    CONST robtarget Target_2200_2:=[[39.025,79.493,0],[0.726314069,0.009187373,0.687236181,-0.009481395],[-2,0,-1,0],[9E+09,9E+09,9E+09,9E+09,9E+09,9E+09]];
    CONST robtarget Target_2210_2:=[[35.542,79.935,0],[0.726314069,0.009187373,0.687236181,-0.009481395],[-2,0,-1,0],[9E+09,9E+09,9E+09,9E+09,9E+09,9E+09]];
    CONST robtarget Target_2220_2:=[[32.97,81.097,0],[0.726314069,0.009187373,0.687236181,-0.009481395],[-2,0,-1,0],[9E+09,9E+09,9E+09,9E+09,9E+09,9E+09]];
    CONST robtarget Target_2230_2:=[[30.756,83.312,0],[0.726314069,0.009187373,0.687236181,-0.009481395],[-2,0,-1,0],[9E+09,9E+09,9E+09,9E+09,9E+09,9E+09]];
    CONST robtarget Target_2240_2:=[[29.841,85.252,0],[0.726314069,0.009187373,0.687236181,-0.009481395],[-2,0,-1,0],[9E+09,9E+09,9E+09,9E+09,9E+09,9E+09]];
    CONST robtarget Target_2250_2:=[[29.28,88.046,0],[0.726314069,0.009187373,0.687236181,-0.009481395],[-2,0,-1,0],[9E+09,9E+09,9E+09,9E+09,9E+09,9E+09]];
    CONST robtarget Target_2260_2:=[[29.205,89.501,0],[0.726314069,0.009187373,0.687236181,-0.009481395],[-2,0,-1,0],[9E+09,9E+09,9E+09,9E+09,9E+09,9E+09]];
    CONST robtarget Target_2270_2:=[[29.324,91.697,0],[0.726314069,0.009187373,0.687236181,-0.009481395],[-2,0,-1,0],[9E+09,9E+09,9E+09,9E+09,9E+09,9E+09]];
    CONST robtarget Target_2280_2:=[[30.172,94.739,0],[0.726314069,0.009187373,0.687236181,-0.009481395],[-2,0,-1,0],[9E+09,9E+09,9E+09,9E+09,9E+09,9E+09]];
    CONST robtarget Target_2290_2:=[[31.657,97.014,0],[0.726314069,0.009187373,0.687236181,-0.009481395],[-2,0,-1,0],[9E+09,9E+09,9E+09,9E+09,9E+09,9E+09]];
    CONST robtarget Target_2300_2:=[[33.883,98.67,0],[0.726314069,0.009187373,0.687236181,-0.009481395],[-2,0,-1,0],[9E+09,9E+09,9E+09,9E+09,9E+09,9E+09]];
    CONST robtarget Target_2310_2:=[[35.769,99.342,0],[0.726314069,0.009187373,0.687236181,-0.009481395],[-2,0,-1,0],[9E+09,9E+09,9E+09,9E+09,9E+09,9E+09]];
    CONST robtarget Target_2320_2:=[[37.808,99.594,0],[0.726314069,0.009187373,0.687236181,-0.009481395],[-2,0,-1,0],[9E+09,9E+09,9E+09,9E+09,9E+09,9E+09]];
    CONST robtarget Target_2330_2:=[[40.664,99.302,0],[0.726314069,0.009187373,0.687236181,-0.009481395],[-2,0,-1,0],[9E+09,9E+09,9E+09,9E+09,9E+09,9E+09]];
    CONST robtarget Target_2340_2:=[[43.731,98.095,0],[0.726314069,0.009187373,0.687236181,-0.009481395],[-2,0,-1,0],[9E+09,9E+09,9E+09,9E+09,9E+09,9E+09]];
    CONST robtarget Target_2350_2:=[[47.413,95.49,0],[0.726314069,0.009187373,0.687236181,-0.009481395],[-2,0,-1,0],[9E+09,9E+09,9E+09,9E+09,9E+09,9E+09]];
    CONST robtarget Target_2360_2:=[[48.093,95.49,0],[0.726314069,0.009187373,0.687236181,-0.009481395],[-2,0,-1,0],[9E+09,9E+09,9E+09,9E+09,9E+09,9E+09]];
    CONST robtarget Target_2370_2:=[[48.093,102.54,0],[0.726314069,0.009187373,0.687236181,-0.009481395],[-2,0,-1,0],[9E+09,9E+09,9E+09,9E+09,9E+09,9E+09]];
    CONST robtarget Target_2380_2:=[[48.093,102.54,10],[0.726314069,0.009187373,0.687236181,-0.009481395],[-2,0,-1,0],[9E+09,9E+09,9E+09,9E+09,9E+09,9E+09]];
    CONST robtarget Target_2390_2:=[[53.685,96.754,10],[0.726314069,0.009187373,0.687236181,-0.009481395],[-2,0,-1,0],[9E+09,9E+09,9E+09,9E+09,9E+09,9E+09]];
    CONST robtarget Target_2400_2:=[[53.685,96.754,0],[0.726314069,0.009187373,0.687236181,-0.009481395],[-2,0,-1,0],[9E+09,9E+09,9E+09,9E+09,9E+09,9E+09]];
    CONST robtarget Target_2410_2:=[[61.781,97.872,0],[0.726314069,0.009187373,0.687236181,-0.009481395],[-2,0,-1,0],[9E+09,9E+09,9E+09,9E+09,9E+09,9E+09]];
    CONST robtarget Target_2420_2:=[[66.233,97.509,0],[0.726314069,0.009187373,0.687236181,-0.009481395],[-2,0,-1,0],[9E+09,9E+09,9E+09,9E+09,9E+09,9E+09]];
    CONST robtarget Target_2430_2:=[[70.243,95.961,0],[0.726314069,0.009187373,0.687236181,-0.009481395],[-2,0,-1,0],[9E+09,9E+09,9E+09,9E+09,9E+09,9E+09]];
    CONST robtarget Target_2440_2:=[[72.614,92.613,0],[0.726314069,0.009187373,0.687236181,-0.009481395],[-2,0,-1,0],[9E+09,9E+09,9E+09,9E+09,9E+09,9E+09]];
    CONST robtarget Target_2450_2:=[[72.964,89.996,0],[0.726314069,0.009187373,0.687236181,-0.009481395],[-2,0,-1,0],[9E+09,9E+09,9E+09,9E+09,9E+09,9E+09]];
    CONST robtarget Target_2460_2:=[[72.964,74.607,0],[0.726314069,0.009187373,0.687236181,-0.009481395],[-2,0,-1,0],[9E+09,9E+09,9E+09,9E+09,9E+09,9E+09]];
    CONST robtarget Target_2470_2:=[[65.962,74.607,0],[0.726314069,0.009187373,0.687236181,-0.009481395],[-2,0,-1,0],[9E+09,9E+09,9E+09,9E+09,9E+09,9E+09]];
    CONST robtarget Target_2480_2:=[[65.962,77.013,0],[0.726314069,0.009187373,0.687236181,-0.009481395],[-2,0,-1,0],[9E+09,9E+09,9E+09,9E+09,9E+09,9E+09]];
    CONST robtarget Target_2490_2:=[[63.118,74.947,0],[0.726314069,0.009187373,0.687236181,-0.009481395],[-2,0,-1,0],[9E+09,9E+09,9E+09,9E+09,9E+09,9E+09]];
    CONST robtarget Target_2500_2:=[[58.766,73.999,0],[0.726314069,0.009187373,0.687236181,-0.009481395],[-2,0,-1,0],[9E+09,9E+09,9E+09,9E+09,9E+09,9E+09]];
    CONST robtarget Target_2510_2:=[[55.832,74.578,0],[0.726314069,0.009187373,0.687236181,-0.009481395],[-2,0,-1,0],[9E+09,9E+09,9E+09,9E+09,9E+09,9E+09]];
    CONST robtarget Target_2520_2:=[[53.483,76.327,0],[0.726314069,0.009187373,0.687236181,-0.009481395],[-2,0,-1,0],[9E+09,9E+09,9E+09,9E+09,9E+09,9E+09]];
    CONST robtarget Target_2530_2:=[[52.081,78.898,0],[0.726314069,0.009187373,0.687236181,-0.009481395],[-2,0,-1,0],[9E+09,9E+09,9E+09,9E+09,9E+09,9E+09]];
    CONST robtarget Target_2540_2:=[[51.789,81.098,0],[0.726314069,0.009187373,0.687236181,-0.009481395],[-2,0,-1,0],[9E+09,9E+09,9E+09,9E+09,9E+09,9E+09]];
    CONST robtarget Target_2550_2:=[[51.983,83.114,0],[0.726314069,0.009187373,0.687236181,-0.009481395],[-2,0,-1,0],[9E+09,9E+09,9E+09,9E+09,9E+09,9E+09]];
    CONST robtarget Target_2560_2:=[[52.864,85.258,0],[0.726314069,0.009187373,0.687236181,-0.009481395],[-2,0,-1,0],[9E+09,9E+09,9E+09,9E+09,9E+09,9E+09]];
    CONST robtarget Target_2570_2:=[[54.039,86.559,0],[0.726314069,0.009187373,0.687236181,-0.009481395],[-2,0,-1,0],[9E+09,9E+09,9E+09,9E+09,9E+09,9E+09]];
    CONST robtarget Target_2580_2:=[[55.703,87.613,0],[0.726314069,0.009187373,0.687236181,-0.009481395],[-2,0,-1,0],[9E+09,9E+09,9E+09,9E+09,9E+09,9E+09]];
    CONST robtarget Target_2590_2:=[[58.542,88.585,0],[0.726314069,0.009187373,0.687236181,-0.009481395],[-2,0,-1,0],[9E+09,9E+09,9E+09,9E+09,9E+09,9E+09]];
    CONST robtarget Target_2600_2:=[[60.612,88.946,0],[0.726314069,0.009187373,0.687236181,-0.009481395],[-2,0,-1,0],[9E+09,9E+09,9E+09,9E+09,9E+09,9E+09]];
    CONST robtarget Target_2610_2:=[[64.587,89.359,0],[0.726314069,0.009187373,0.687236181,-0.009481395],[-2,0,-1,0],[9E+09,9E+09,9E+09,9E+09,9E+09,9E+09]];
    CONST robtarget Target_2620_2:=[[66.011,89.461,0],[0.726314069,0.009187373,0.687236181,-0.009481395],[-2,0,-1,0],[9E+09,9E+09,9E+09,9E+09,9E+09,9E+09]];
    CONST robtarget Target_2630_2:=[[66.011,89.582,0],[0.726314069,0.009187373,0.687236181,-0.009481395],[-2,0,-1,0],[9E+09,9E+09,9E+09,9E+09,9E+09,9E+09]];
    CONST robtarget Target_2640_2:=[[64.625,92.171,0],[0.726314069,0.009187373,0.687236181,-0.009481395],[-2,0,-1,0],[9E+09,9E+09,9E+09,9E+09,9E+09,9E+09]];
    CONST robtarget Target_2650_2:=[[60.468,92.889,0],[0.726314069,0.009187373,0.687236181,-0.009481395],[-2,0,-1,0],[9E+09,9E+09,9E+09,9E+09,9E+09,9E+09]];
    CONST robtarget Target_2660_2:=[[54.293,91.284,0],[0.726314069,0.009187373,0.687236181,-0.009481395],[-2,0,-1,0],[9E+09,9E+09,9E+09,9E+09,9E+09,9E+09]];
    CONST robtarget Target_2670_2:=[[53.685,91.284,0],[0.726314069,0.009187373,0.687236181,-0.009481395],[-2,0,-1,0],[9E+09,9E+09,9E+09,9E+09,9E+09,9E+09]];
    CONST robtarget Target_2680_2:=[[53.685,96.754,0],[0.726314069,0.009187373,0.687236181,-0.009481395],[-2,0,-1,0],[9E+09,9E+09,9E+09,9E+09,9E+09,9E+09]];
    CONST robtarget Target_2690_2:=[[53.685,96.754,10],[0.726314069,0.009187373,0.687236181,-0.009481395],[-2,0,-1,0],[9E+09,9E+09,9E+09,9E+09,9E+09,9E+09]];
    CONST robtarget Target_2700_2:=[[65.962,85.206,10],[0.726314069,0.009187373,0.687236181,-0.009481395],[-2,0,-1,0],[9E+09,9E+09,9E+09,9E+09,9E+09,9E+09]];
    CONST robtarget Target_2710_2:=[[65.962,85.206,0],[0.726314069,0.009187373,0.687236181,-0.009481395],[-2,0,-1,0],[9E+09,9E+09,9E+09,9E+09,9E+09,9E+09]];
    CONST robtarget Target_2720_2:=[[60.881,84.38,0],[0.726314069,0.009187373,0.687236181,-0.009481395],[-2,0,-1,0],[9E+09,9E+09,9E+09,9E+09,9E+09,9E+09]];
    CONST robtarget Target_2730_2:=[[59.422,83.407,0],[0.726314069,0.009187373,0.687236181,-0.009481395],[-2,0,-1,0],[9E+09,9E+09,9E+09,9E+09,9E+09,9E+09]];
    CONST robtarget Target_2740_2:=[[58.912,81.681,0],[0.726314069,0.009187373,0.687236181,-0.009481395],[-2,0,-1,0],[9E+09,9E+09,9E+09,9E+09,9E+09,9E+09]];
    CONST robtarget Target_2750_2:=[[59.032,80.639,0],[0.726314069,0.009187373,0.687236181,-0.009481395],[-2,0,-1,0],[9E+09,9E+09,9E+09,9E+09,9E+09,9E+09]];
    CONST robtarget Target_2760_2:=[[60.054,79.339,0],[0.726314069,0.009187373,0.687236181,-0.009481395],[-2,0,-1,0],[9E+09,9E+09,9E+09,9E+09,9E+09,9E+09]];
    CONST robtarget Target_2770_2:=[[61.465,78.954,0],[0.726314069,0.009187373,0.687236181,-0.009481395],[-2,0,-1,0],[9E+09,9E+09,9E+09,9E+09,9E+09,9E+09]];
    CONST robtarget Target_2780_2:=[[62.315,78.91,0],[0.726314069,0.009187373,0.687236181,-0.009481395],[-2,0,-1,0],[9E+09,9E+09,9E+09,9E+09,9E+09,9E+09]];
    CONST robtarget Target_2790_2:=[[64.212,79.335,0],[0.726314069,0.009187373,0.687236181,-0.009481395],[-2,0,-1,0],[9E+09,9E+09,9E+09,9E+09,9E+09,9E+09]];
    CONST robtarget Target_2800_2:=[[65.962,80.514,0],[0.726314069,0.009187373,0.687236181,-0.009481395],[-2,0,-1,0],[9E+09,9E+09,9E+09,9E+09,9E+09,9E+09]];
    CONST robtarget Target_2810_2:=[[65.962,85.206,0],[0.726314069,0.009187373,0.687236181,-0.009481395],[-2,0,-1,0],[9E+09,9E+09,9E+09,9E+09,9E+09,9E+09]];
    CONST robtarget Target_2820_2:=[[65.962,85.206,10],[0.726314069,0.009187373,0.687236181,-0.009481395],[-2,0,-1,0],[9E+09,9E+09,9E+09,9E+09,9E+09,9E+09]];
    CONST robtarget Target_2830_2:=[[78.191,105.944,10],[0.726314069,0.009187373,0.687236181,-0.009481395],[-2,0,-1,0],[9E+09,9E+09,9E+09,9E+09,9E+09,9E+09]];
    CONST robtarget Target_2840_2:=[[78.191,105.944,0],[0.726314069,0.009187373,0.687236181,-0.009481395],[-2,0,-1,0],[9E+09,9E+09,9E+09,9E+09,9E+09,9E+09]];
    CONST robtarget Target_2850_2:=[[78.191,74.607,0],[0.726314069,0.009187373,0.687236181,-0.009481395],[-2,0,-1,0],[9E+09,9E+09,9E+09,9E+09,9E+09,9E+09]];
    CONST robtarget Target_2860_2:=[[84.949,74.607,0],[0.726314069,0.009187373,0.687236181,-0.009481395],[-1,0,-1,0],[9E+09,9E+09,9E+09,9E+09,9E+09,9E+09]];
    CONST robtarget Target_2870_2:=[[85.241,75.725,0],[0.726314069,0.009187373,0.687236181,-0.009481395],[-1,0,-1,0],[9E+09,9E+09,9E+09,9E+09,9E+09,9E+09]];
    CONST robtarget Target_2880_2:=[[90.832,74.169,0],[0.726314069,0.009187373,0.687236181,-0.009481395],[-1,0,-1,0],[9E+09,9E+09,9E+09,9E+09,9E+09,9E+09]];
    CONST robtarget Target_2890_2:=[[94.512,74.978,0],[0.726314069,0.009187373,0.687236181,-0.009481395],[-1,0,-1,0],[9E+09,9E+09,9E+09,9E+09,9E+09,9E+09]];
    CONST robtarget Target_2900_2:=[[97.536,77.39,0],[0.726314069,0.009187373,0.687236181,-0.009481395],[-1,-1,0,0],[9E+09,9E+09,9E+09,9E+09,9E+09,9E+09]];
    CONST robtarget Target_2910_2:=[[99.251,80.187,0],[0.726314069,0.009187373,0.687236181,-0.009481395],[-1,-1,0,0],[9E+09,9E+09,9E+09,9E+09,9E+09,9E+09]];
    CONST robtarget Target_2920_2:=[[100.173,83.531,0],[0.726314069,0.009187373,0.687236181,-0.009481395],[-1,-1,0,0],[9E+09,9E+09,9E+09,9E+09,9E+09,9E+09]];
    CONST robtarget Target_2930_2:=[[100.362,86.227,0],[0.726314069,0.009187373,0.687236181,-0.009481395],[-1,-1,0,0],[9E+09,9E+09,9E+09,9E+09,9E+09,9E+09]];
    CONST robtarget Target_2940_2:=[[100.162,89.348,0],[0.726314069,0.009187373,0.687236181,-0.009481395],[-1,-1,0,0],[9E+09,9E+09,9E+09,9E+09,9E+09,9E+09]];
    CONST robtarget Target_2950_2:=[[99.451,92.348,0],[0.726314069,0.009187373,0.687236181,-0.009481395],[-1,-1,0,0],[9E+09,9E+09,9E+09,9E+09,9E+09,9E+09]];
    CONST robtarget Target_2960_2:=[[98.126,94.909,0],[0.726314069,0.009187373,0.687236181,-0.009481395],[-1,-1,0,0],[9E+09,9E+09,9E+09,9E+09,9E+09,9E+09]];
    CONST robtarget Target_2970_2:=[[96.145,96.789,0],[0.726314069,0.009187373,0.687236181,-0.009481395],[-1,0,-1,0],[9E+09,9E+09,9E+09,9E+09,9E+09,9E+09]];
    CONST robtarget Target_2980_2:=[[93.246,97.782,0],[0.726314069,0.009187373,0.687236181,-0.009481395],[-1,0,-1,0],[9E+09,9E+09,9E+09,9E+09,9E+09,9E+09]];
    CONST robtarget Target_2990_2:=[[91.056,97.792,0],[0.726314069,0.009187373,0.687236181,-0.009481395],[-1,0,-1,0],[9E+09,9E+09,9E+09,9E+09,9E+09,9E+09]];
    CONST robtarget Target_3000_2:=[[88.708,97.17,0],[0.726314069,0.009187373,0.687236181,-0.009481395],[-1,0,-1,0],[9E+09,9E+09,9E+09,9E+09,9E+09,9E+09]];
    CONST robtarget Target_3010_2:=[[86.849,96.094,0],[0.726314069,0.009187373,0.687236181,-0.009481395],[-1,0,-1,0],[9E+09,9E+09,9E+09,9E+09,9E+09,9E+09]];
    CONST robtarget Target_3020_2:=[[85.241,94.858,0],[0.726314069,0.009187373,0.687236181,-0.009481395],[-1,0,-1,0],[9E+09,9E+09,9E+09,9E+09,9E+09,9E+09]];
    CONST robtarget Target_3030_2:=[[85.241,105.944,0],[0.726314069,0.009187373,0.687236181,-0.009481395],[-1,0,-1,0],[9E+09,9E+09,9E+09,9E+09,9E+09,9E+09]];
    CONST robtarget Target_3040_2:=[[78.191,105.944,0],[0.726314069,0.009187373,0.687236181,-0.009481395],[-2,0,-1,0],[9E+09,9E+09,9E+09,9E+09,9E+09,9E+09]];
    CONST robtarget Target_3050_2:=[[78.191,105.944,10],[0.726314069,0.009187373,0.687236181,-0.009481395],[-2,0,-1,0],[9E+09,9E+09,9E+09,9E+09,9E+09,9E+09]];
    CONST robtarget Target_3060_2:=[[85.241,91.138,10],[0.726314069,0.009187373,0.687236181,-0.009481395],[-1,0,-1,0],[9E+09,9E+09,9E+09,9E+09,9E+09,9E+09]];
    CONST robtarget Target_3070_2:=[[85.241,91.138,0],[0.726314069,0.009187373,0.687236181,-0.009481395],[-1,0,-1,0],[9E+09,9E+09,9E+09,9E+09,9E+09,9E+09]];
    CONST robtarget Target_3080_2:=[[85.241,79.809,0],[0.726314069,0.009187373,0.687236181,-0.009481395],[-1,0,-1,0],[9E+09,9E+09,9E+09,9E+09,9E+09,9E+09]];
    CONST robtarget Target_3090_2:=[[88.085,79.323,0],[0.726314069,0.009187373,0.687236181,-0.009481395],[-1,0,-1,0],[9E+09,9E+09,9E+09,9E+09,9E+09,9E+09]];
    CONST robtarget Target_3100_2:=[[90.106,79.66,0],[0.726314069,0.009187373,0.687236181,-0.009481395],[-1,0,-1,0],[9E+09,9E+09,9E+09,9E+09,9E+09,9E+09]];
    CONST robtarget Target_3110_2:=[[91.905,81.033,0],[0.726314069,0.009187373,0.687236181,-0.009481395],[-1,0,-1,0],[9E+09,9E+09,9E+09,9E+09,9E+09,9E+09]];
    CONST robtarget Target_3120_2:=[[92.891,83.394,0],[0.726314069,0.009187373,0.687236181,-0.009481395],[-1,0,-1,0],[9E+09,9E+09,9E+09,9E+09,9E+09,9E+09]];
    CONST robtarget Target_3130_2:=[[93.142,86.082,0],[0.726314069,0.009187373,0.687236181,-0.009481395],[-1,0,-1,0],[9E+09,9E+09,9E+09,9E+09,9E+09,9E+09]];
    CONST robtarget Target_3140_2:=[[92.957,88.611,0],[0.726314069,0.009187373,0.687236181,-0.009481395],[-1,0,-1,0],[9E+09,9E+09,9E+09,9E+09,9E+09,9E+09]];
    CONST robtarget Target_3150_2:=[[92.311,90.605,0],[0.726314069,0.009187373,0.687236181,-0.009481395],[-1,0,-1,0],[9E+09,9E+09,9E+09,9E+09,9E+09,9E+09]];
    CONST robtarget Target_3160_2:=[[90.724,92.035,0],[0.726314069,0.009187373,0.687236181,-0.009481395],[-1,0,-1,0],[9E+09,9E+09,9E+09,9E+09,9E+09,9E+09]];
    CONST robtarget Target_3170_2:=[[88.961,92.354,0],[0.726314069,0.009187373,0.687236181,-0.009481395],[-1,0,-1,0],[9E+09,9E+09,9E+09,9E+09,9E+09,9E+09]];
    CONST robtarget Target_3180_2:=[[87.176,92.081,0],[0.726314069,0.009187373,0.687236181,-0.009481395],[-1,0,-1,0],[9E+09,9E+09,9E+09,9E+09,9E+09,9E+09]];
    CONST robtarget Target_3190_2:=[[85.241,91.138,0],[0.726314069,0.009187373,0.687236181,-0.009481395],[-1,0,-1,0],[9E+09,9E+09,9E+09,9E+09,9E+09,9E+09]];
    CONST robtarget Target_3200_2:=[[85.241,91.138,10],[0.726314069,0.009187373,0.687236181,-0.009481395],[-1,0,-1,0],[9E+09,9E+09,9E+09,9E+09,9E+09,9E+09]];
    CONST robtarget Target_3210_2:=[[114.293,92.889,10],[0.726314069,0.009187373,0.687236181,-0.009481395],[-1,-1,0,0],[9E+09,9E+09,9E+09,9E+09,9E+09,9E+09]];
    CONST robtarget Target_3220_2:=[[114.293,92.889,0],[0.726314069,0.009187373,0.687236181,-0.009481395],[-1,-1,0,0],[9E+09,9E+09,9E+09,9E+09,9E+09,9E+09]];
    CONST robtarget Target_3230_2:=[[111.516,91.894,0],[0.726314069,0.009187373,0.687236181,-0.009481395],[-1,-1,0,0],[9E+09,9E+09,9E+09,9E+09,9E+09,9E+09]];
    CONST robtarget Target_3240_2:=[[110.079,88.878,0],[0.726314069,0.009187373,0.687236181,-0.009481395],[-1,-1,0,0],[9E+09,9E+09,9E+09,9E+09,9E+09,9E+09]];
    CONST robtarget Target_3250_2:=[[109.82,85.731,0],[0.726314069,0.009187373,0.687236181,-0.009481395],[-1,-1,0,0],[9E+09,9E+09,9E+09,9E+09,9E+09,9E+09]];
    CONST robtarget Target_3260_2:=[[110.134,82.622,0],[0.726314069,0.009187373,0.687236181,-0.009481395],[-1,-1,0,0],[9E+09,9E+09,9E+09,9E+09,9E+09,9E+09]];
    CONST robtarget Target_3270_2:=[[112.748,79.215,0],[0.726314069,0.009187373,0.687236181,-0.009481395],[-1,-1,0,0],[9E+09,9E+09,9E+09,9E+09,9E+09,9E+09]];
    CONST robtarget Target_3280_2:=[[115.472,79.116,0],[0.726314069,0.009187373,0.687236181,-0.009481395],[-1,-1,0,0],[9E+09,9E+09,9E+09,9E+09,9E+09,9E+09]];
    CONST robtarget Target_3290_2:=[[117.853,81.029,0],[0.726314069,0.009187373,0.687236181,-0.009481395],[-1,-1,0,0],[9E+09,9E+09,9E+09,9E+09,9E+09,9E+09]];
    CONST robtarget Target_3300_2:=[[118.692,84.329,0],[0.726314069,0.009187373,0.687236181,-0.009481395],[-1,-1,0,0],[9E+09,9E+09,9E+09,9E+09,9E+09,9E+09]];
    CONST robtarget Target_3310_2:=[[118.705,87.144,0],[0.726314069,0.009187373,0.687236181,-0.009481395],[-1,-1,0,0],[9E+09,9E+09,9E+09,9E+09,9E+09,9E+09]];
    CONST robtarget Target_3320_2:=[[117.699,91.082,0],[0.726314069,0.009187373,0.687236181,-0.009481395],[-1,-1,0,0],[9E+09,9E+09,9E+09,9E+09,9E+09,9E+09]];
    CONST robtarget Target_3330_2:=[[116.9,92.042,0],[0.726314069,0.009187373,0.687236181,-0.009481395],[-1,-1,0,0],[9E+09,9E+09,9E+09,9E+09,9E+09,9E+09]];
    CONST robtarget Target_3340_2:=[[114.293,92.889,0],[0.726314069,0.009187373,0.687236181,-0.009481395],[-1,-1,0,0],[9E+09,9E+09,9E+09,9E+09,9E+09,9E+09]];
    CONST robtarget Target_3350_2:=[[114.293,92.889,10],[0.726314069,0.009187373,0.687236181,-0.009481395],[-1,-1,0,0],[9E+09,9E+09,9E+09,9E+09,9E+09,9E+09]];
    CONST robtarget Target_3360_2:=[[114.293,97.945,10],[0.726314069,0.009187373,0.687236181,-0.009481395],[-1,-1,0,0],[9E+09,9E+09,9E+09,9E+09,9E+09,9E+09]];
    CONST robtarget Target_3370_2:=[[114.293,97.945,0],[0.726314069,0.009187373,0.687236181,-0.009481395],[-1,-1,0,0],[9E+09,9E+09,9E+09,9E+09,9E+09,9E+09]];
    CONST robtarget Target_3380_2:=[[119.425,97.063,0],[0.726314069,0.009187373,0.687236181,-0.009481395],[-1,-1,0,0],[9E+09,9E+09,9E+09,9E+09,9E+09,9E+09]];
    CONST robtarget Target_3390_2:=[[122.854,94.783,0],[0.726314069,0.009187373,0.687236181,-0.009481395],[-1,-1,0,0],[9E+09,9E+09,9E+09,9E+09,9E+09,9E+09]];
    CONST robtarget Target_3400_2:=[[124.981,91.496,0],[0.726314069,0.009187373,0.687236181,-0.009481395],[-1,-1,0,0],[9E+09,9E+09,9E+09,9E+09,9E+09,9E+09]];
    CONST robtarget Target_3410_2:=[[125.918,87.222,0],[0.726314069,0.009187373,0.687236181,-0.009481395],[-1,-1,0,0],[9E+09,9E+09,9E+09,9E+09,9E+09,9E+09]];
    CONST robtarget Target_3420_2:=[[125.74,83.065,0],[0.726314069,0.009187373,0.687236181,-0.009481395],[-1,-1,0,0],[9E+09,9E+09,9E+09,9E+09,9E+09,9E+09]];
    CONST robtarget Target_3430_2:=[[124.292,78.941,0],[0.726314069,0.009187373,0.687236181,-0.009481395],[-1,-1,0,0],[9E+09,9E+09,9E+09,9E+09,9E+09,9E+09]];
    CONST robtarget Target_3440_2:=[[122.614,76.811,0],[0.726314069,0.009187373,0.687236181,-0.009481395],[-1,-1,0,0],[9E+09,9E+09,9E+09,9E+09,9E+09,9E+09]];
    CONST robtarget Target_3450_2:=[[118.869,74.576,0],[0.726314069,0.009187373,0.687236181,-0.009481395],[-1,-1,0,0],[9E+09,9E+09,9E+09,9E+09,9E+09,9E+09]];
    CONST robtarget Target_3460_2:=[[115.671,73.954,0],[0.726314069,0.009187373,0.687236181,-0.009481395],[-1,-1,0,0],[9E+09,9E+09,9E+09,9E+09,9E+09,9E+09]];
    CONST robtarget Target_3470_2:=[[111.694,74.099,0],[0.726314069,0.009187373,0.687236181,-0.009481395],[-1,-1,0,0],[9E+09,9E+09,9E+09,9E+09,9E+09,9E+09]];
    CONST robtarget Target_3480_2:=[[107.574,75.575,0],[0.726314069,0.009187373,0.687236181,-0.009481395],[-1,-1,0,0],[9E+09,9E+09,9E+09,9E+09,9E+09,9E+09]];
    CONST robtarget Target_3490_2:=[[104.577,78.476,0],[0.726314069,0.009187373,0.687236181,-0.009481395],[-1,-1,0,0],[9E+09,9E+09,9E+09,9E+09,9E+09,9E+09]];
    CONST robtarget Target_3500_2:=[[103.102,81.78,0],[0.726314069,0.009187373,0.687236181,-0.009481395],[-1,-1,0,0],[9E+09,9E+09,9E+09,9E+09,9E+09,9E+09]];
    CONST robtarget Target_3510_2:=[[102.673,84.234,0],[0.726314069,0.009187373,0.687236181,-0.009481395],[-1,-1,0,0],[9E+09,9E+09,9E+09,9E+09,9E+09,9E+09]];
    CONST robtarget Target_3520_2:=[[102.712,87.979,0],[0.726314069,0.009187373,0.687236181,-0.009481395],[-1,-1,0,0],[9E+09,9E+09,9E+09,9E+09,9E+09,9E+09]];
    CONST robtarget Target_3530_2:=[[103.395,91.017,0],[0.726314069,0.009187373,0.687236181,-0.009481395],[-1,-1,0,0],[9E+09,9E+09,9E+09,9E+09,9E+09,9E+09]];
    CONST robtarget Target_3540_2:=[[104.511,93.286,0],[0.726314069,0.009187373,0.687236181,-0.009481395],[-1,-1,0,0],[9E+09,9E+09,9E+09,9E+09,9E+09,9E+09]];
    CONST robtarget Target_3550_2:=[[106.651,95.634,0],[0.726314069,0.009187373,0.687236181,-0.009481395],[-1,-1,0,0],[9E+09,9E+09,9E+09,9E+09,9E+09,9E+09]];
    CONST robtarget Target_3560_2:=[[109.412,97.163,0],[0.726314069,0.009187373,0.687236181,-0.009481395],[-1,-1,0,0],[9E+09,9E+09,9E+09,9E+09,9E+09,9E+09]];
    CONST robtarget Target_3570_2:=[[114.293,97.945,0],[0.726314069,0.009187373,0.687236181,-0.009481395],[-1,-1,0,0],[9E+09,9E+09,9E+09,9E+09,9E+09,9E+09]];
    CONST robtarget Target_3580_2:=[[114.293,97.945,10],[0.726314069,0.009187373,0.687236181,-0.009481395],[-1,-1,0,0],[9E+09,9E+09,9E+09,9E+09,9E+09,9E+09]];
    CONST robtarget Target_3590_2:=[[57.132,66.1,10],[0.726314069,0.009187373,0.687236181,-0.009481395],[-2,0,-1,0],[9E+09,9E+09,9E+09,9E+09,9E+09,9E+09]];
    CONST robtarget Target_3600_2:=[[57.132,66.1,0],[0.726314069,0.009187373,0.687236181,-0.009481395],[-2,0,-1,0],[9E+09,9E+09,9E+09,9E+09,9E+09,9E+09]];
    CONST robtarget Target_3610_2:=[[40.852,48.713,0],[0.726314069,0.009187373,0.687236181,-0.009481395],[-2,0,-1,0],[9E+09,9E+09,9E+09,9E+09,9E+09,9E+09]];
    CONST robtarget Target_3620_2:=[[40.852,45.296,0],[0.726314069,0.009187373,0.687236181,-0.009481395],[-2,0,-1,0],[9E+09,9E+09,9E+09,9E+09,9E+09,9E+09]];
    CONST robtarget Target_3630_2:=[[75,4.113,0],[0.726314069,0.009187373,0.687236181,-0.009481395],[-2,0,-1,0],[9E+09,9E+09,9E+09,9E+09,9E+09,9E+09]];
    CONST robtarget Target_3640_2:=[[109.148,45.296,0],[0.726314069,0.009187373,0.687236181,-0.009481395],[-1,-1,0,0],[9E+09,9E+09,9E+09,9E+09,9E+09,9E+09]];
    CONST robtarget Target_3650_2:=[[109.148,48.713,0],[0.726314069,0.009187373,0.687236181,-0.009481395],[-1,-1,0,0],[9E+09,9E+09,9E+09,9E+09,9E+09,9E+09]];
    CONST robtarget Target_3660_2:=[[92.868,66.1,0],[0.726314069,0.009187373,0.687236181,-0.009481395],[-1,0,-1,0],[9E+09,9E+09,9E+09,9E+09,9E+09,9E+09]];
    CONST robtarget Target_3670_2:=[[57.132,66.1,0],[0.726314069,0.009187373,0.687236181,-0.009481395],[-2,0,-1,0],[9E+09,9E+09,9E+09,9E+09,9E+09,9E+09]];
    CONST robtarget Target_3680_2:=[[57.132,66.1,10],[0.726314069,0.009187373,0.687236181,-0.009481395],[-2,0,-1,0],[9E+09,9E+09,9E+09,9E+09,9E+09,9E+09]];
    CONST robtarget Target_3690_2:=[[59.3,61.1,10],[0.726314069,0.009187373,0.687236181,-0.009481395],[-2,0,-1,0],[9E+09,9E+09,9E+09,9E+09,9E+09,9E+09]];
    CONST robtarget Target_3700_2:=[[59.3,61.1,0],[0.726314069,0.009187373,0.687236181,-0.009481395],[-2,0,-1,0],[9E+09,9E+09,9E+09,9E+09,9E+09,9E+09]];
    CONST robtarget Target_3710_2:=[[48.446,49.508,0],[0.726314069,0.009187373,0.687236181,-0.009481395],[-2,0,-1,0],[9E+09,9E+09,9E+09,9E+09,9E+09,9E+09]];
    CONST robtarget Target_3720_2:=[[59.481,49.508,0],[0.726314069,0.009187373,0.687236181,-0.009481395],[-2,0,-1,0],[9E+09,9E+09,9E+09,9E+09,9E+09,9E+09]];
    CONST robtarget Target_3730_2:=[[69.526,61.1,0],[0.726314069,0.009187373,0.687236181,-0.009481395],[-2,0,-1,0],[9E+09,9E+09,9E+09,9E+09,9E+09,9E+09]];
    CONST robtarget Target_3740_2:=[[59.3,61.1,0],[0.726314069,0.009187373,0.687236181,-0.009481395],[-2,0,-1,0],[9E+09,9E+09,9E+09,9E+09,9E+09,9E+09]];
    CONST robtarget Target_3750_2:=[[59.3,61.1,10],[0.726314069,0.009187373,0.687236181,-0.009481395],[-2,0,-1,0],[9E+09,9E+09,9E+09,9E+09,9E+09,9E+09]];
    CONST robtarget Target_3760_2:=[[80.474,61.1,10],[0.726314069,0.009187373,0.687236181,-0.009481395],[-2,0,-1,0],[9E+09,9E+09,9E+09,9E+09,9E+09,9E+09]];
    CONST robtarget Target_3770_2:=[[80.474,61.1,0],[0.726314069,0.009187373,0.687236181,-0.009481395],[-2,0,-1,0],[9E+09,9E+09,9E+09,9E+09,9E+09,9E+09]];
    CONST robtarget Target_3780_2:=[[90.7,61.1,0],[0.726314069,0.009187373,0.687236181,-0.009481395],[-1,0,-1,0],[9E+09,9E+09,9E+09,9E+09,9E+09,9E+09]];
    CONST robtarget Target_3790_2:=[[101.554,49.508,0],[0.726314069,0.009187373,0.687236181,-0.009481395],[-1,-1,0,0],[9E+09,9E+09,9E+09,9E+09,9E+09,9E+09]];
    CONST robtarget Target_3800_2:=[[90.519,49.508,0],[0.726314069,0.009187373,0.687236181,-0.009481395],[-1,0,-1,0],[9E+09,9E+09,9E+09,9E+09,9E+09,9E+09]];
    CONST robtarget Target_3810_2:=[[80.474,61.1,0],[0.726314069,0.009187373,0.687236181,-0.009481395],[-2,0,-1,0],[9E+09,9E+09,9E+09,9E+09,9E+09,9E+09]];
    CONST robtarget Target_3820_2:=[[80.474,61.1,10],[0.726314069,0.009187373,0.687236181,-0.009481395],[-2,0,-1,0],[9E+09,9E+09,9E+09,9E+09,9E+09,9E+09]];
    CONST robtarget Target_3830_2:=[[75,59.782,10],[0.726314069,0.009187373,0.687236181,-0.009481395],[-2,0,-1,0],[9E+09,9E+09,9E+09,9E+09,9E+09,9E+09]];
    CONST robtarget Target_3840_2:=[[75,59.782,0],[0.726314069,0.009187373,0.687236181,-0.009481395],[-2,0,-1,0],[9E+09,9E+09,9E+09,9E+09,9E+09,9E+09]];
    CONST robtarget Target_3850_2:=[[83.903,49.508,0],[0.726314069,0.009187373,0.687236181,-0.009481395],[-1,0,-1,0],[9E+09,9E+09,9E+09,9E+09,9E+09,9E+09]];
    CONST robtarget Target_3860_2:=[[66.097,49.508,0],[0.726314069,0.009187373,0.687236181,-0.009481395],[-2,0,-1,0],[9E+09,9E+09,9E+09,9E+09,9E+09,9E+09]];
    CONST robtarget Target_3870_2:=[[75,59.782,0],[0.726314069,0.009187373,0.687236181,-0.009481395],[-2,0,-1,0],[9E+09,9E+09,9E+09,9E+09,9E+09,9E+09]];
    CONST robtarget Target_3880_2:=[[75,59.782,10],[0.726314069,0.009187373,0.687236181,-0.009481395],[-2,0,-1,0],[9E+09,9E+09,9E+09,9E+09,9E+09,9E+09]];
    CONST robtarget Target_3890_2:=[[64.21,44.508,10],[0.726314069,0.009187373,0.687236181,-0.009481395],[-2,0,-1,0],[9E+09,9E+09,9E+09,9E+09,9E+09,9E+09]];
    CONST robtarget Target_3900_2:=[[64.21,44.508,0],[0.726314069,0.009187373,0.687236181,-0.009481395],[-2,0,-1,0],[9E+09,9E+09,9E+09,9E+09,9E+09,9E+09]];
    CONST robtarget Target_3910_2:=[[85.79,44.508,0],[0.726314069,0.009187373,0.687236181,-0.009481395],[-1,0,-1,0],[9E+09,9E+09,9E+09,9E+09,9E+09,9E+09]];
    CONST robtarget Target_3920_2:=[[75,15.254,0],[0.726314069,0.009187373,0.687236181,-0.009481395],[-2,0,-1,0],[9E+09,9E+09,9E+09,9E+09,9E+09,9E+09]];
    CONST robtarget Target_3930_2:=[[64.21,44.508,0],[0.726314069,0.009187373,0.687236181,-0.009481395],[-2,0,-1,0],[9E+09,9E+09,9E+09,9E+09,9E+09,9E+09]];
    CONST robtarget Target_3940_2:=[[64.21,44.508,10],[0.726314069,0.009187373,0.687236181,-0.009481395],[-2,0,-1,0],[9E+09,9E+09,9E+09,9E+09,9E+09,9E+09]];
    CONST robtarget Target_3950_2:=[[58.88,44.508,10],[0.726314069,0.009187373,0.687236181,-0.009481395],[-2,0,-1,0],[9E+09,9E+09,9E+09,9E+09,9E+09,9E+09]];
    CONST robtarget Target_3960_2:=[[58.88,44.508,0],[0.726314069,0.009187373,0.687236181,-0.009481395],[-2,0,-1,0],[9E+09,9E+09,9E+09,9E+09,9E+09,9E+09]];
    CONST robtarget Target_3970_2:=[[48.001,44.508,0],[0.726314069,0.009187373,0.687236181,-0.009481395],[-2,0,-1,0],[9E+09,9E+09,9E+09,9E+09,9E+09,9E+09]];
    CONST robtarget Target_3980_2:=[[67.598,20.874,0],[0.726314069,0.009187373,0.687236181,-0.009481395],[-2,0,-1,0],[9E+09,9E+09,9E+09,9E+09,9E+09,9E+09]];
    CONST robtarget Target_3990_2:=[[58.88,44.508,0],[0.726314069,0.009187373,0.687236181,-0.009481395],[-2,0,-1,0],[9E+09,9E+09,9E+09,9E+09,9E+09,9E+09]];
    CONST robtarget Target_4000_2:=[[58.88,44.508,10],[0.726314069,0.009187373,0.687236181,-0.009481395],[-2,0,-1,0],[9E+09,9E+09,9E+09,9E+09,9E+09,9E+09]];
    CONST robtarget Target_4010_2:=[[91.12,44.508,10],[0.726314069,0.009187373,0.687236181,-0.009481395],[-1,0,-1,0],[9E+09,9E+09,9E+09,9E+09,9E+09,9E+09]];
    CONST robtarget Target_4020_2:=[[91.12,44.508,0],[0.726314069,0.009187373,0.687236181,-0.009481395],[-1,0,-1,0],[9E+09,9E+09,9E+09,9E+09,9E+09,9E+09]];
    CONST robtarget Target_4030_2:=[[101.999,44.508,0],[0.726314069,0.009187373,0.687236181,-0.009481395],[-1,-1,0,0],[9E+09,9E+09,9E+09,9E+09,9E+09,9E+09]];
    CONST robtarget Target_4040_2:=[[82.402,20.874,0],[0.726314069,0.009187373,0.687236181,-0.009481395],[-1,0,-1,0],[9E+09,9E+09,9E+09,9E+09,9E+09,9E+09]];
    CONST robtarget Target_4050_2:=[[91.12,44.508,0],[0.726314069,0.009187373,0.687236181,-0.009481395],[-1,0,-1,0],[9E+09,9E+09,9E+09,9E+09,9E+09,9E+09]];
    CONST robtarget Target_Home_Espejo:=[[-676.754166789,677.141454372,-133.14230978],[0.358218118,-0.604139007,0.620387065,0.349021104],[-1,0,-1,0],[9E+09,9E+09,9E+09,9E+09,9E+09,9E+09]];
!Ejercicio hecho en clase
    !TASK PERS wobjdata wcaja:=[FALSE,TRUE,"",[[-78.3768,-694.538,672.47],[0.999913,-0.00011372,0.00016022,0.0132033]],[[-74.9038,-552.314,679.445],[0.0262226,-0.999656,6.92619E-06,1.8063E-05]]];
    !***********************************************************
    !
    ! M?dulo:  Module1
    !
    ! Descripción:
    !   <Introduzca la descripción aquí>
    !
    ! Autor: GabrielBojaca y Mafe Morillo
    !
    ! Versión: 1.0
    !
    !***********************************************************


    !***********************************************************
    !
    ! Procedimiento Main
    !
    !   Este es el punto de entrada de su programa
    !
    !***********************************************************
    PROC main()
        !MoveAbsJ Home_ABS, v1000, z1, tool0;
        !Path_10;
        MoveAbsJ Home_ABS, v300, z1, tool0;

        TPErase;
        TPWrite "INICIO PROGRAMA";
        TPWrite "APAGADO BANDA TRANASPORTADORA";
        Reset DO_02;
        Reset DO_01;
        RESET BWD_Conveyor;
        RESET FWD_Conveyor;

        WHILE TRUE DO
            IF DI_03 = 1 THEN
                RESET BWD_Conveyor;
                Reset FWD_Conveyor;
                Set BWD_Conveyor;
                WaitTime 2;
                Reset FWD_Conveyor;
                Reset BWD_Conveyor;
            ENDIF

            IF DI_01 = 1 AND DI_02 = 0 THEN
                TPWrite "ENCIENDE BANDA TRANASPORTADORA";
                Set FWD_Conveyor;
                WaitTime 2.03;  !2.05 el mejor hasta ahora
                TPWrite "APAGADO BANDA TRANASPORTADORA";
                Reset FWD_Conveyor;
                TPWrite "INICIANDO DECORADO";
                Set DO_01;
                Path_10;
                TPWrite "DECORADO FINALIZADO";
                Reset DO_01;
                MoveAbsJ Home_ABS,v1000,z1,tool0;
                TPWrite "ENCENDIDO BANDA TRANASPORTADORA";
                Set FWD_Conveyor;
                WaitTime 8;
                TPWrite "APAGADO BANDA TRANASPORTADORA";
                Reset FWD_Conveyor;

            ELSEIF DI_01 = 0 AND DI_02=1 THEN
                Set DO_02;
                TPWrite "RUTINA CAMBIO DE HERRAMIENTA";
                MoveAbsJ Mantenimiento_Point,v1000,z1,tool0;
                TPWrite "PELIGRO";
                TPWrite "OPERARIO CERCA A HERRAMIENTA";
                TPWrite "PRESIONE LOS DOS BOTONES PARA CONTINUAR EL PROGRAMA";
                WaitDI DI_01,1;
                WaitDI DI_02,1;
                Reset DO_02;
                TPWrite "REANUDANDO PROGRAMA";
                WaitTime 3;
                MoveAbsJ Home_ABS,v1000,z1,tool0;
            ELSEIF DI_01 = 0 AND DI_02=0 THEN
                TPWrite "ESPERANDO INSTRUCCIÓNES";
            ELSEIF DI_01 = 1 AND DI_02=1 THEN
                TPWrite "ERROR";
                TPWrite "NO DEBE PRESIONAR AMBAS ENTRADAS AL TIEMPO";
            ENDIF

        ENDWHILE



    ENDPROC

    PROC Test_Caja()
        RESET BWD_Conveyor;
        Reset FWD_Conveyor;
        Set BWD_Conveyor;
        WaitTime 2;
        Reset FWD_Conveyor;
        Reset BWD_Conveyor;
    ENDPROC

    PROC Aristas_Caja()
        MoveL Target_10,v1000,z1,Marcador_TCP\WObj:=Caja;
        MoveL Target_20,v1000,z1,Marcador_TCP\WObj:=Caja;
        MoveL Target_30,v1000,z1,Marcador_TCP\WObj:=Caja;
        MoveL Target_40,v1000,z1,Marcador_TCP\WObj:=Caja;
    ENDPROC
    PROC MAFE()

    ENDPROC
    PROC Path_10()
        MoveL Home_cafe,v1000,z1,Marcador_TCP\WObj:=Caja;
        MoveL Target_60,v1000,z1,Marcador_TCP\WObj:=Caja;
        MoveL Target_70,v1000,z1,Marcador_TCP\WObj:=Caja;
        MoveL Target_80,v1000,z1,Marcador_TCP\WObj:=Caja;
        MoveL Target_90,v1000,z1,Marcador_TCP\WObj:=Caja;
        MoveL Target_100,v1000,z1,Marcador_TCP\WObj:=Caja;
        MoveL Target_110,v1000,z1,Marcador_TCP\WObj:=Caja;
        MoveL Target_120,v1000,z1,Marcador_TCP\WObj:=Caja;
        MoveL Target_130,v1000,z1,Marcador_TCP\WObj:=Caja;
        MoveL Target_140,v1000,z1,Marcador_TCP\WObj:=Caja;
        MoveL Target_150,v1000,z1,Marcador_TCP\WObj:=Caja;
        MoveL Target_160,v1000,z1,Marcador_TCP\WObj:=Caja;
        MoveL Target_170,v1000,z1,Marcador_TCP\WObj:=Caja;
        MoveL Target_180,v1000,z1,Marcador_TCP\WObj:=Caja;
        MoveL Target_190,v1000,z1,Marcador_TCP\WObj:=Caja;
        MoveL Target_200,v1000,z1,Marcador_TCP\WObj:=Caja;
        MoveL Target_210,v1000,z1,Marcador_TCP\WObj:=Caja;
        MoveL Target_220,v1000,z1,Marcador_TCP\WObj:=Caja;
        MoveL Target_230,v1000,z1,Marcador_TCP\WObj:=Caja;
        MoveL Target_240,v1000,z1,Marcador_TCP\WObj:=Caja;
        MoveL Target_250,v1000,z1,Marcador_TCP\WObj:=Caja;
        MoveL Target_260,v1000,z1,Marcador_TCP\WObj:=Caja;
        MoveL Target_270,v1000,z1,Marcador_TCP\WObj:=Caja;
        MoveL Target_280,v1000,z1,Marcador_TCP\WObj:=Caja;
        MoveL Target_290,v1000,z1,Marcador_TCP\WObj:=Caja;
        MoveL Target_300,v1000,z1,Marcador_TCP\WObj:=Caja;
        MoveL Target_310,v1000,z1,Marcador_TCP\WObj:=Caja;
        MoveL Target_320,v1000,z1,Marcador_TCP\WObj:=Caja;
        MoveL Target_330,v1000,z1,Marcador_TCP\WObj:=Caja;
        MoveL Target_340,v1000,z1,Marcador_TCP\WObj:=Caja;
        MoveL Target_350,v1000,z1,Marcador_TCP\WObj:=Caja;
        MoveL Target_360,v1000,z1,Marcador_TCP\WObj:=Caja;
        MoveL Target_370,v1000,z1,Marcador_TCP\WObj:=Caja;
        MoveL Target_380,v1000,z1,Marcador_TCP\WObj:=Caja;
        MoveL Target_390,v1000,z1,Marcador_TCP\WObj:=Caja;
        MoveL Target_400,v1000,z1,Marcador_TCP\WObj:=Caja;
        MoveL Target_410,v1000,z1,Marcador_TCP\WObj:=Caja;
        MoveL Target_420,v1000,z1,Marcador_TCP\WObj:=Caja;
        MoveL Target_430,v1000,z1,Marcador_TCP\WObj:=Caja;
        MoveL Target_440,v1000,z1,Marcador_TCP\WObj:=Caja;
        MoveL Target_450,v1000,z1,Marcador_TCP\WObj:=Caja;
        MoveL Target_460,v1000,z1,Marcador_TCP\WObj:=Caja;
        MoveL Target_470,v1000,z1,Marcador_TCP\WObj:=Caja;
        MoveL Target_480,v1000,z1,Marcador_TCP\WObj:=Caja;
        MoveL Target_490,v1000,z1,Marcador_TCP\WObj:=Caja;
        MoveL Target_500,v1000,z1,Marcador_TCP\WObj:=Caja;
        MoveL Target_510,v1000,z1,Marcador_TCP\WObj:=Caja;
        MoveL Target_520,v1000,z1,Marcador_TCP\WObj:=Caja;
        MoveL Target_530,v1000,z1,Marcador_TCP\WObj:=Caja;
        MoveL Target_540,v1000,z1,Marcador_TCP\WObj:=Caja;
        MoveL Target_550,v1000,z1,Marcador_TCP\WObj:=Caja;
        MoveL Target_560,v1000,z1,Marcador_TCP\WObj:=Caja;
        MoveL Target_570,v1000,z1,Marcador_TCP\WObj:=Caja;
        MoveL Target_580,v1000,z1,Marcador_TCP\WObj:=Caja;
        MoveL Target_590,v1000,z1,Marcador_TCP\WObj:=Caja;
        MoveL Target_600,v1000,z1,Marcador_TCP\WObj:=Caja;
        MoveL Target_610,v1000,z1,Marcador_TCP\WObj:=Caja;
        MoveL Target_620,v1000,z1,Marcador_TCP\WObj:=Caja;
        MoveL Target_630,v1000,z1,Marcador_TCP\WObj:=Caja;
        MoveL Target_640,v1000,z1,Marcador_TCP\WObj:=Caja;
        MoveL Target_650,v1000,z1,Marcador_TCP\WObj:=Caja;
        MoveL Target_660,v1000,z1,Marcador_TCP\WObj:=Caja;
        MoveL Target_670,v1000,z1,Marcador_TCP\WObj:=Caja;
        MoveL Target_680,v1000,z1,Marcador_TCP\WObj:=Caja;
        MoveL Target_690,v1000,z1,Marcador_TCP\WObj:=Caja;
        MoveL Target_700,v1000,z1,Marcador_TCP\WObj:=Caja;
        MoveL Target_710,v1000,z1,Marcador_TCP\WObj:=Caja;
        MoveL Target_720,v1000,z1,Marcador_TCP\WObj:=Caja;
        MoveL Target_730,v1000,z1,Marcador_TCP\WObj:=Caja;
        MoveL Target_740,v1000,z1,Marcador_TCP\WObj:=Caja;
        MoveL Target_750,v1000,z1,Marcador_TCP\WObj:=Caja;
        MoveL Target_760,v1000,z1,Marcador_TCP\WObj:=Caja;
        MoveL Target_770,v1000,z1,Marcador_TCP\WObj:=Caja;
        MoveL Target_780,v1000,z1,Marcador_TCP\WObj:=Caja;
        MoveL Target_790,v1000,z1,Marcador_TCP\WObj:=Caja;
        MoveL Target_800,v1000,z1,Marcador_TCP\WObj:=Caja;
        MoveL Target_810,v1000,z1,Marcador_TCP\WObj:=Caja;
        MoveL Target_820,v1000,z1,Marcador_TCP\WObj:=Caja;
        MoveL Target_830,v1000,z1,Marcador_TCP\WObj:=Caja;
        MoveL Target_840,v1000,z1,Marcador_TCP\WObj:=Caja;
        MoveL Target_850,v1000,z1,Marcador_TCP\WObj:=Caja;
        MoveL Target_860,v1000,z1,Marcador_TCP\WObj:=Caja;
        MoveL Target_870,v1000,z1,Marcador_TCP\WObj:=Caja;
        MoveL Target_880,v1000,z1,Marcador_TCP\WObj:=Caja;
        MoveL Target_890,v1000,z1,Marcador_TCP\WObj:=Caja;
        MoveL Target_900,v1000,z1,Marcador_TCP\WObj:=Caja;
        MoveL Target_910,v1000,z1,Marcador_TCP\WObj:=Caja;
        MoveL Target_920,v1000,z1,Marcador_TCP\WObj:=Caja;
        MoveL Target_930,v1000,z1,Marcador_TCP\WObj:=Caja;
        MoveL Target_940,v1000,z1,Marcador_TCP\WObj:=Caja;
        MoveL Target_950,v1000,z1,Marcador_TCP\WObj:=Caja;
        MoveL Target_960,v1000,z1,Marcador_TCP\WObj:=Caja;
        MoveL Target_970,v1000,z1,Marcador_TCP\WObj:=Caja;
        MoveL Target_980,v1000,z1,Marcador_TCP\WObj:=Caja;
        MoveL Target_990,v1000,z1,Marcador_TCP\WObj:=Caja;
        MoveL Target_1000,v1000,z1,Marcador_TCP\WObj:=Caja;
        MoveL Target_1010,v1000,z1,Marcador_TCP\WObj:=Caja;
        MoveL Target_1020,v1000,z1,Marcador_TCP\WObj:=Caja;
        MoveL Target_1030,v1000,z1,Marcador_TCP\WObj:=Caja;
        MoveL Target_1040,v1000,z1,Marcador_TCP\WObj:=Caja;
        MoveL Target_1050,v1000,z1,Marcador_TCP\WObj:=Caja;
        MoveL Target_1060,v1000,z1,Marcador_TCP\WObj:=Caja;
        MoveL Target_1070,v1000,z1,Marcador_TCP\WObj:=Caja;
        MoveL Target_1080,v1000,z1,Marcador_TCP\WObj:=Caja;
        MoveL Target_1090,v1000,z1,Marcador_TCP\WObj:=Caja;
        MoveL Target_1100,v1000,z1,Marcador_TCP\WObj:=Caja;
        MoveL Target_1110,v1000,z1,Marcador_TCP\WObj:=Caja;
        MoveL Target_1120,v1000,z1,Marcador_TCP\WObj:=Caja;
        MoveL Target_1130,v1000,z1,Marcador_TCP\WObj:=Caja;
        MoveL Target_1140,v1000,z1,Marcador_TCP\WObj:=Caja;
        MoveL Target_1150,v1000,z1,Marcador_TCP\WObj:=Caja;
        MoveL Target_1160,v1000,z1,Marcador_TCP\WObj:=Caja;
        MoveL Target_1170,v1000,z1,Marcador_TCP\WObj:=Caja;
        MoveL Target_1180,v1000,z1,Marcador_TCP\WObj:=Caja;
        MoveL Target_1190,v1000,z1,Marcador_TCP\WObj:=Caja;
        MoveL Target_1200,v1000,z1,Marcador_TCP\WObj:=Caja;
        MoveL Target_1210,v1000,z1,Marcador_TCP\WObj:=Caja;
        MoveL Target_1220,v1000,z1,Marcador_TCP\WObj:=Caja;
        MoveL Target_1230,v1000,z1,Marcador_TCP\WObj:=Caja;
        MoveL Target_1240,v1000,z1,Marcador_TCP\WObj:=Caja;
        MoveL Target_1250,v1000,z1,Marcador_TCP\WObj:=Caja;
        MoveL Target_1260,v1000,z1,Marcador_TCP\WObj:=Caja;
        MoveL Target_1270,v1000,z1,Marcador_TCP\WObj:=Caja;
        MoveL Target_1280,v1000,z1,Marcador_TCP\WObj:=Caja;
        MoveL Target_1290,v1000,z1,Marcador_TCP\WObj:=Caja;
        MoveL Target_1300,v1000,z1,Marcador_TCP\WObj:=Caja;
        MoveL Target_1310,v1000,z1,Marcador_TCP\WObj:=Caja;
        MoveL Target_1320,v1000,z1,Marcador_TCP\WObj:=Caja;
        MoveL Target_1330,v1000,z1,Marcador_TCP\WObj:=Caja;
        MoveL Target_1340,v1000,z1,Marcador_TCP\WObj:=Caja;
        MoveL Target_1350,v1000,z1,Marcador_TCP\WObj:=Caja;
        MoveL Target_1360,v1000,z1,Marcador_TCP\WObj:=Caja;
        MoveL Target_1370,v1000,z1,Marcador_TCP\WObj:=Caja;
        MoveL Target_1380,v1000,z1,Marcador_TCP\WObj:=Caja;
        MoveL Target_1390,v1000,z1,Marcador_TCP\WObj:=Caja;
        MoveL Target_1400,v1000,z1,Marcador_TCP\WObj:=Caja;
        MoveL Target_1410,v1000,z1,Marcador_TCP\WObj:=Caja;
        MoveL Target_1420,v1000,z1,Marcador_TCP\WObj:=Caja;
        MoveL Target_1430,v1000,z1,Marcador_TCP\WObj:=Caja;
        MoveL Target_1440,v1000,z1,Marcador_TCP\WObj:=Caja;
        MoveL Target_1450,v1000,z1,Marcador_TCP\WObj:=Caja;
        MoveL Target_1460,v1000,z1,Marcador_TCP\WObj:=Caja;
        MoveL Target_1470,v1000,z1,Marcador_TCP\WObj:=Caja;
        MoveL Target_1480,v1000,z1,Marcador_TCP\WObj:=Caja;
        MoveL Target_1490,v1000,z1,Marcador_TCP\WObj:=Caja;
        MoveL Target_1500,v1000,z1,Marcador_TCP\WObj:=Caja;
        MoveL Target_1510,v1000,z1,Marcador_TCP\WObj:=Caja;
        MoveL Target_1520,v1000,z1,Marcador_TCP\WObj:=Caja;
        MoveL Target_1530,v1000,z1,Marcador_TCP\WObj:=Caja;
        MoveL Target_1540,v1000,z1,Marcador_TCP\WObj:=Caja;
        MoveL Target_1550,v1000,z1,Marcador_TCP\WObj:=Caja;
        MoveL Target_1560,v1000,z1,Marcador_TCP\WObj:=Caja;
        MoveL Target_1570,v1000,z1,Marcador_TCP\WObj:=Caja;
        MoveL Target_1580,v1000,z1,Marcador_TCP\WObj:=Caja;
        MoveL Target_1590,v1000,z1,Marcador_TCP\WObj:=Caja;
        MoveL Target_1600,v1000,z1,Marcador_TCP\WObj:=Caja;
        MoveL Target_1610,v1000,z1,Marcador_TCP\WObj:=Caja;
        MoveL Target_1620,v1000,z1,Marcador_TCP\WObj:=Caja;
        MoveL Target_1630,v1000,z1,Marcador_TCP\WObj:=Caja;
        MoveL Target_1640,v1000,z1,Marcador_TCP\WObj:=Caja;
        MoveL Target_1650,v1000,z1,Marcador_TCP\WObj:=Caja;
        MoveL Target_1660,v1000,z1,Marcador_TCP\WObj:=Caja;
        MoveL Target_1670,v1000,z1,Marcador_TCP\WObj:=Caja;
        MoveL Target_1680,v1000,z1,Marcador_TCP\WObj:=Caja;
        MoveL Target_1690,v1000,z1,Marcador_TCP\WObj:=Caja;
        MoveL Target_1700,v1000,z1,Marcador_TCP\WObj:=Caja;
        MoveL Target_1710,v1000,z1,Marcador_TCP\WObj:=Caja;
        MoveL Target_1720,v1000,z1,Marcador_TCP\WObj:=Caja;
        MoveL Target_1730,v1000,z1,Marcador_TCP\WObj:=Caja;
        MoveL Target_1740,v1000,z1,Marcador_TCP\WObj:=Caja;
        MoveL Target_1750,v1000,z1,Marcador_TCP\WObj:=Caja;
        MoveL Target_1760,v1000,z1,Marcador_TCP\WObj:=Caja;
        MoveL Target_1770,v1000,z1,Marcador_TCP\WObj:=Caja;
        MoveL Target_1780,v1000,z1,Marcador_TCP\WObj:=Caja;
        MoveL Target_1790,v1000,z1,Marcador_TCP\WObj:=Caja;
        MoveL Target_1800,v1000,z1,Marcador_TCP\WObj:=Caja;
        MoveL Target_1810,v1000,z1,Marcador_TCP\WObj:=Caja;
        MoveL Target_1820,v1000,z1,Marcador_TCP\WObj:=Caja;
        MoveL Target_1830,v1000,z1,Marcador_TCP\WObj:=Caja;
        MoveL Target_1840,v1000,z1,Marcador_TCP\WObj:=Caja;
        MoveL Target_1850,v1000,z1,Marcador_TCP\WObj:=Caja;
        MoveL Target_1860,v1000,z1,Marcador_TCP\WObj:=Caja;
        MoveL Target_1870,v1000,z1,Marcador_TCP\WObj:=Caja;
        MoveL Target_1880,v1000,z1,Marcador_TCP\WObj:=Caja;
        MoveL Target_1890,v1000,z1,Marcador_TCP\WObj:=Caja;
        MoveL Target_1900,v1000,z1,Marcador_TCP\WObj:=Caja;
        MoveL Target_1910,v1000,z1,Marcador_TCP\WObj:=Caja;
        MoveL Target_1920,v1000,z1,Marcador_TCP\WObj:=Caja;
        MoveL Target_1930,v1000,z1,Marcador_TCP\WObj:=Caja;
        MoveL Target_1940,v1000,z1,Marcador_TCP\WObj:=Caja;
        MoveL Target_1950,v1000,z1,Marcador_TCP\WObj:=Caja;
        MoveL Target_1960,v1000,z1,Marcador_TCP\WObj:=Caja;
        MoveL Target_1970,v1000,z1,Marcador_TCP\WObj:=Caja;
        MoveL Target_1980,v1000,z1,Marcador_TCP\WObj:=Caja;
        MoveL Target_1990,v1000,z1,Marcador_TCP\WObj:=Caja;
        MoveL Target_2000,v1000,z1,Marcador_TCP\WObj:=Caja;
        MoveL Target_2010,v1000,z1,Marcador_TCP\WObj:=Caja;
        MoveL Target_2020,v1000,z1,Marcador_TCP\WObj:=Caja;
        MoveL Target_2030,v1000,z1,Marcador_TCP\WObj:=Caja;
        MoveL Target_2040,v1000,z1,Marcador_TCP\WObj:=Caja;
        MoveL Target_2050,v1000,z1,Marcador_TCP\WObj:=Caja;
        MoveL Target_2060,v1000,z1,Marcador_TCP\WObj:=Caja;
        MoveL Target_2070,v1000,z1,Marcador_TCP\WObj:=Caja;
        MoveL Target_2080,v1000,z1,Marcador_TCP\WObj:=Caja;
        MoveL Target_2090,v1000,z1,Marcador_TCP\WObj:=Caja;
        MoveL Target_2100,v1000,z1,Marcador_TCP\WObj:=Caja;
        MoveL Target_2110,v1000,z1,Marcador_TCP\WObj:=Caja;
        MoveL Target_2120,v1000,z1,Marcador_TCP\WObj:=Caja;
        MoveL Target_2130,v1000,z1,Marcador_TCP\WObj:=Caja;
        MoveL Target_2140,v1000,z1,Marcador_TCP\WObj:=Caja;
        MoveL Target_2150,v1000,z1,Marcador_TCP\WObj:=Caja;
        MoveL Target_2160,v1000,z1,Marcador_TCP\WObj:=Caja;
        MoveL Target_2170,v1000,z1,Marcador_TCP\WObj:=Caja;
        MoveL Target_2180,v1000,z1,Marcador_TCP\WObj:=Caja;
        MoveL Target_2190,v1000,z1,Marcador_TCP\WObj:=Caja;
        MoveL Target_2200,v1000,z1,Marcador_TCP\WObj:=Caja;
        MoveL Target_2210,v1000,z1,Marcador_TCP\WObj:=Caja;
        MoveL Target_2220,v1000,z1,Marcador_TCP\WObj:=Caja;
        MoveL Target_2230,v1000,z1,Marcador_TCP\WObj:=Caja;
        MoveL Target_2240,v1000,z1,Marcador_TCP\WObj:=Caja;
        MoveL Target_2250,v1000,z1,Marcador_TCP\WObj:=Caja;
        MoveL Target_2260,v1000,z1,Marcador_TCP\WObj:=Caja;
        MoveL Target_2270,v1000,z1,Marcador_TCP\WObj:=Caja;
        MoveL Target_2280,v1000,z1,Marcador_TCP\WObj:=Caja;
        MoveL Target_2290,v1000,z1,Marcador_TCP\WObj:=Caja;
        MoveL Target_2300,v1000,z1,Marcador_TCP\WObj:=Caja;
        MoveL Target_2310,v1000,z1,Marcador_TCP\WObj:=Caja;
        MoveL Target_2320,v1000,z1,Marcador_TCP\WObj:=Caja;
        MoveL Target_2330,v1000,z1,Marcador_TCP\WObj:=Caja;
        MoveL Target_2340,v1000,z1,Marcador_TCP\WObj:=Caja;
        MoveL Target_2350,v1000,z1,Marcador_TCP\WObj:=Caja;
        MoveL Target_2360,v1000,z1,Marcador_TCP\WObj:=Caja;
        MoveL Target_2370,v1000,z1,Marcador_TCP\WObj:=Caja;
        MoveL Target_2380,v1000,z1,Marcador_TCP\WObj:=Caja;
        MoveL Target_2390,v1000,z1,Marcador_TCP\WObj:=Caja;
        MoveL Target_2400,v1000,z1,Marcador_TCP\WObj:=Caja;
        MoveL Target_2410,v1000,z1,Marcador_TCP\WObj:=Caja;
        MoveL Target_2420,v1000,z1,Marcador_TCP\WObj:=Caja;
        MoveL Target_2430,v1000,z1,Marcador_TCP\WObj:=Caja;
        MoveL Target_2440,v1000,z1,Marcador_TCP\WObj:=Caja;
        MoveL Target_2450,v1000,z1,Marcador_TCP\WObj:=Caja;
        MoveL Target_2460,v1000,z1,Marcador_TCP\WObj:=Caja;
        MoveL Target_2470,v1000,z1,Marcador_TCP\WObj:=Caja;
        MoveL Target_2480,v1000,z1,Marcador_TCP\WObj:=Caja;
        MoveL Target_2490,v1000,z1,Marcador_TCP\WObj:=Caja;
        MoveL Target_2500,v1000,z1,Marcador_TCP\WObj:=Caja;
        MoveL Target_2510,v1000,z1,Marcador_TCP\WObj:=Caja;
        MoveL Target_2520,v1000,z1,Marcador_TCP\WObj:=Caja;
        MoveL Target_2530,v1000,z1,Marcador_TCP\WObj:=Caja;
        MoveL Target_2540,v1000,z1,Marcador_TCP\WObj:=Caja;
        MoveL Target_2550,v1000,z1,Marcador_TCP\WObj:=Caja;
        MoveL Target_2560,v1000,z1,Marcador_TCP\WObj:=Caja;
        MoveL Target_2570,v1000,z1,Marcador_TCP\WObj:=Caja;
        MoveL Target_2580,v1000,z1,Marcador_TCP\WObj:=Caja;
        MoveL Target_2590,v1000,z1,Marcador_TCP\WObj:=Caja;
        MoveL Target_2600,v1000,z1,Marcador_TCP\WObj:=Caja;
        MoveL Target_2610,v1000,z1,Marcador_TCP\WObj:=Caja;
        MoveL Target_2620,v1000,z1,Marcador_TCP\WObj:=Caja;
        MoveL Target_2630,v1000,z1,Marcador_TCP\WObj:=Caja;
        MoveL Target_2640,v1000,z1,Marcador_TCP\WObj:=Caja;
        MoveL Target_2650,v1000,z1,Marcador_TCP\WObj:=Caja;
        MoveL Target_2660,v1000,z1,Marcador_TCP\WObj:=Caja;
        MoveL Target_2670,v1000,z1,Marcador_TCP\WObj:=Caja;
        MoveL Target_2680,v1000,z1,Marcador_TCP\WObj:=Caja;
        MoveL Target_2690,v1000,z1,Marcador_TCP\WObj:=Caja;
        MoveL Target_2700,v1000,z1,Marcador_TCP\WObj:=Caja;
        MoveL Target_2710,v1000,z1,Marcador_TCP\WObj:=Caja;
        MoveL Target_2720,v1000,z1,Marcador_TCP\WObj:=Caja;
        MoveL Target_2730,v1000,z1,Marcador_TCP\WObj:=Caja;
        MoveL Target_2740,v1000,z1,Marcador_TCP\WObj:=Caja;
        MoveL Target_2750,v1000,z1,Marcador_TCP\WObj:=Caja;
        MoveL Target_2760,v1000,z1,Marcador_TCP\WObj:=Caja;
        MoveL Target_2770,v1000,z1,Marcador_TCP\WObj:=Caja;
        MoveL Target_2780,v1000,z1,Marcador_TCP\WObj:=Caja;
        MoveL Target_2790,v1000,z1,Marcador_TCP\WObj:=Caja;
        MoveL Target_2800,v1000,z1,Marcador_TCP\WObj:=Caja;
        MoveL Target_2810,v1000,z1,Marcador_TCP\WObj:=Caja;
        MoveL Target_2820,v1000,z1,Marcador_TCP\WObj:=Caja;
        MoveL Target_2830,v1000,z1,Marcador_TCP\WObj:=Caja;
        MoveL Target_2840,v1000,z1,Marcador_TCP\WObj:=Caja;
        MoveL Target_2850,v1000,z1,Marcador_TCP\WObj:=Caja;
        MoveL Target_2860,v1000,z1,Marcador_TCP\WObj:=Caja;
        MoveL Target_2870,v1000,z1,Marcador_TCP\WObj:=Caja;
        MoveL Target_2880,v1000,z1,Marcador_TCP\WObj:=Caja;
        MoveL Target_2890,v1000,z1,Marcador_TCP\WObj:=Caja;
        MoveL Target_2900,v1000,z1,Marcador_TCP\WObj:=Caja;
        MoveL Target_2910,v1000,z1,Marcador_TCP\WObj:=Caja;
        MoveL Target_2920,v1000,z1,Marcador_TCP\WObj:=Caja;
        MoveL Target_2930,v1000,z1,Marcador_TCP\WObj:=Caja;
        MoveL Target_2940,v1000,z1,Marcador_TCP\WObj:=Caja;
        MoveL Target_2950,v1000,z1,Marcador_TCP\WObj:=Caja;
        MoveL Target_2960,v1000,z1,Marcador_TCP\WObj:=Caja;
        MoveL Target_2970,v1000,z1,Marcador_TCP\WObj:=Caja;
        MoveL Target_2980,v1000,z1,Marcador_TCP\WObj:=Caja;
        MoveL Target_2990,v1000,z1,Marcador_TCP\WObj:=Caja;
        MoveL Target_3000,v1000,z1,Marcador_TCP\WObj:=Caja;
        MoveL Target_3010,v1000,z1,Marcador_TCP\WObj:=Caja;
        MoveL Target_3020,v1000,z1,Marcador_TCP\WObj:=Caja;
        MoveL Target_3030,v1000,z1,Marcador_TCP\WObj:=Caja;
        MoveL Target_3040,v1000,z1,Marcador_TCP\WObj:=Caja;
        MoveL Target_3050,v1000,z1,Marcador_TCP\WObj:=Caja;
        MoveL Target_3060,v1000,z1,Marcador_TCP\WObj:=Caja;
        MoveL Target_3070,v1000,z1,Marcador_TCP\WObj:=Caja;
        MoveL Target_3080,v1000,z1,Marcador_TCP\WObj:=Caja;
        MoveL Target_3090,v1000,z1,Marcador_TCP\WObj:=Caja;
        MoveL Target_3100,v1000,z1,Marcador_TCP\WObj:=Caja;
        MoveL Target_3110,v1000,z1,Marcador_TCP\WObj:=Caja;
        MoveL Target_3120,v1000,z1,Marcador_TCP\WObj:=Caja;
        MoveL Target_3130,v1000,z1,Marcador_TCP\WObj:=Caja;
        MoveL Target_3140,v1000,z1,Marcador_TCP\WObj:=Caja;
        MoveL Target_3150,v1000,z1,Marcador_TCP\WObj:=Caja;
        MoveL Target_3160,v1000,z1,Marcador_TCP\WObj:=Caja;
        MoveL Target_3170,v1000,z1,Marcador_TCP\WObj:=Caja;
        MoveL Target_3180,v1000,z1,Marcador_TCP\WObj:=Caja;
        MoveL Target_3190,v1000,z1,Marcador_TCP\WObj:=Caja;
        MoveL Target_3200,v1000,z1,Marcador_TCP\WObj:=Caja;
        MoveL Target_3210,v1000,z1,Marcador_TCP\WObj:=Caja;
        MoveL Target_3220,v1000,z1,Marcador_TCP\WObj:=Caja;
        MoveL Target_3230,v1000,z1,Marcador_TCP\WObj:=Caja;
        MoveL Target_3240,v1000,z1,Marcador_TCP\WObj:=Caja;
        MoveL Target_3250,v1000,z1,Marcador_TCP\WObj:=Caja;
        MoveL Target_3260,v1000,z1,Marcador_TCP\WObj:=Caja;
        MoveL Target_3270,v1000,z1,Marcador_TCP\WObj:=Caja;
        MoveL Target_3280,v1000,z1,Marcador_TCP\WObj:=Caja;
        MoveL Target_3290,v1000,z1,Marcador_TCP\WObj:=Caja;
        MoveL Target_3300,v1000,z1,Marcador_TCP\WObj:=Caja;
        MoveL Target_3310,v1000,z1,Marcador_TCP\WObj:=Caja;
        MoveL Target_3320,v1000,z1,Marcador_TCP\WObj:=Caja;
        MoveL Target_3330,v1000,z1,Marcador_TCP\WObj:=Caja;
        MoveL Target_3340,v1000,z1,Marcador_TCP\WObj:=Caja;
        MoveL Target_3350,v1000,z1,Marcador_TCP\WObj:=Caja;
        MoveL Target_3360,v1000,z1,Marcador_TCP\WObj:=Caja;
        MoveL Target_3370,v1000,z1,Marcador_TCP\WObj:=Caja;
        MoveL Target_3380,v1000,z1,Marcador_TCP\WObj:=Caja;
        MoveL Target_3390,v1000,z1,Marcador_TCP\WObj:=Caja;
        MoveL Target_3400,v1000,z1,Marcador_TCP\WObj:=Caja;
        MoveL Target_3410,v1000,z1,Marcador_TCP\WObj:=Caja;
        MoveL Target_3420,v1000,z1,Marcador_TCP\WObj:=Caja;
        MoveL Target_3430,v1000,z1,Marcador_TCP\WObj:=Caja;
        MoveL Target_3440,v1000,z1,Marcador_TCP\WObj:=Caja;
        MoveL Target_3450,v1000,z1,Marcador_TCP\WObj:=Caja;
        MoveL Target_3460,v1000,z1,Marcador_TCP\WObj:=Caja;
        MoveL Target_3470,v1000,z1,Marcador_TCP\WObj:=Caja;
        MoveL Target_3480,v1000,z1,Marcador_TCP\WObj:=Caja;
        MoveL Target_3490,v1000,z1,Marcador_TCP\WObj:=Caja;
        MoveL Target_3500,v1000,z1,Marcador_TCP\WObj:=Caja;
        MoveL Target_3510,v1000,z1,Marcador_TCP\WObj:=Caja;
        MoveL Target_3520,v1000,z1,Marcador_TCP\WObj:=Caja;
        MoveL Target_3530,v1000,z1,Marcador_TCP\WObj:=Caja;
        MoveL Target_3540,v1000,z1,Marcador_TCP\WObj:=Caja;
        MoveL Target_3550,v1000,z1,Marcador_TCP\WObj:=Caja;
        MoveL Target_3560,v1000,z1,Marcador_TCP\WObj:=Caja;
        MoveL Target_3570,v1000,z1,Marcador_TCP\WObj:=Caja;
        MoveL Target_3580,v1000,z1,Marcador_TCP\WObj:=Caja;
        MoveL Target_3590,v1000,z1,Marcador_TCP\WObj:=Caja;
        MoveL Target_3600,v1000,z1,Marcador_TCP\WObj:=Caja;
        MoveL Target_3610,v1000,z1,Marcador_TCP\WObj:=Caja;
        MoveL Target_3620,v1000,z1,Marcador_TCP\WObj:=Caja;
        MoveL Target_3630,v1000,z1,Marcador_TCP\WObj:=Caja;
        MoveL Target_3640,v1000,z1,Marcador_TCP\WObj:=Caja;
        MoveL Target_3650,v1000,z1,Marcador_TCP\WObj:=Caja;
        MoveL Target_3660,v1000,z1,Marcador_TCP\WObj:=Caja;
        MoveL Target_3670,v1000,z1,Marcador_TCP\WObj:=Caja;
        MoveL Target_3680,v1000,z1,Marcador_TCP\WObj:=Caja;
        MoveL Target_3690,v1000,z1,Marcador_TCP\WObj:=Caja;
        MoveL Target_3700,v1000,z1,Marcador_TCP\WObj:=Caja;
        MoveL Target_3710,v1000,z1,Marcador_TCP\WObj:=Caja;
        MoveL Target_3720,v1000,z1,Marcador_TCP\WObj:=Caja;
        MoveL Target_3730,v1000,z1,Marcador_TCP\WObj:=Caja;
        MoveL Target_3740,v1000,z1,Marcador_TCP\WObj:=Caja;
        MoveL Target_3750,v1000,z1,Marcador_TCP\WObj:=Caja;
        MoveL Target_3760,v1000,z1,Marcador_TCP\WObj:=Caja;
        MoveL Target_3770,v1000,z1,Marcador_TCP\WObj:=Caja;
        MoveL Target_3780,v1000,z1,Marcador_TCP\WObj:=Caja;
        MoveL Target_3790,v1000,z1,Marcador_TCP\WObj:=Caja;
        MoveL Target_3800,v1000,z1,Marcador_TCP\WObj:=Caja;
        MoveL Target_3810,v1000,z1,Marcador_TCP\WObj:=Caja;
        MoveL Target_3820,v1000,z1,Marcador_TCP\WObj:=Caja;
        MoveL Target_3830,v1000,z1,Marcador_TCP\WObj:=Caja;
        MoveL Target_3840,v1000,z1,Marcador_TCP\WObj:=Caja;
        MoveL Target_3850,v1000,z1,Marcador_TCP\WObj:=Caja;
        MoveL Target_3860,v1000,z1,Marcador_TCP\WObj:=Caja;
        MoveL Target_3870,v1000,z1,Marcador_TCP\WObj:=Caja;
        MoveL Target_3880,v1000,z1,Marcador_TCP\WObj:=Caja;
        MoveL Target_3890,v1000,z1,Marcador_TCP\WObj:=Caja;
        MoveL Target_3900,v1000,z1,Marcador_TCP\WObj:=Caja;
        MoveL Target_3910,v1000,z1,Marcador_TCP\WObj:=Caja;
        MoveL Target_3920,v1000,z1,Marcador_TCP\WObj:=Caja;
        MoveL Target_3930,v1000,z1,Marcador_TCP\WObj:=Caja;
        MoveL Target_3940,v1000,z1,Marcador_TCP\WObj:=Caja;
        MoveL Target_3950,v1000,z1,Marcador_TCP\WObj:=Caja;
        MoveL Target_3960,v1000,z1,Marcador_TCP\WObj:=Caja;
        MoveL Target_3970,v1000,z1,Marcador_TCP\WObj:=Caja;
        MoveL Target_3980,v1000,z1,Marcador_TCP\WObj:=Caja;
        MoveL Target_3990,v1000,z1,Marcador_TCP\WObj:=Caja;
        MoveL Target_4000,v1000,z1,Marcador_TCP\WObj:=Caja;
        MoveL Target_4010,v1000,z1,Marcador_TCP\WObj:=Caja;
        MoveL Target_4020,v1000,z1,Marcador_TCP\WObj:=Caja;
        MoveL Target_4030,v1000,z1,Marcador_TCP\WObj:=Caja;
        MoveL Target_4040,v1000,z1,Marcador_TCP\WObj:=Caja;
        MoveL Target_4050,v1000,z1,Marcador_TCP\WObj:=Caja;
        MoveL Target_4060,v1000,z1,Marcador_TCP\WObj:=Caja;
        MoveL Home_cafe,v1000,z1,Marcador_TCP\WObj:=Caja;
    ENDPROC
    PROC Path_Espejo()
        MoveL Target_Home_Espejo,v1000,z1,Marcador_TCP\WObj:=Caja_2;
        MoveL Home_cafe_2,v1000,z1,Marcador_TCP\WObj:=Caja_2;
        MoveL Target_60_2,v1000,z1,Marcador_TCP\WObj:=Caja_2;
        MoveL Target_70_2,v1000,z1,Marcador_TCP\WObj:=Caja_2;
        MoveL Target_80_2,v1000,z1,Marcador_TCP\WObj:=Caja_2;
        MoveL Target_90_2,v1000,z1,Marcador_TCP\WObj:=Caja_2;
        MoveL Target_100_2,v1000,z1,Marcador_TCP\WObj:=Caja_2;
        MoveL Target_110_2,v1000,z1,Marcador_TCP\WObj:=Caja_2;
        MoveL Target_120_2,v1000,z1,Marcador_TCP\WObj:=Caja_2;
        MoveL Target_130_2,v1000,z1,Marcador_TCP\WObj:=Caja_2;
        MoveL Target_140_2,v1000,z1,Marcador_TCP\WObj:=Caja_2;
        MoveL Target_150_2,v1000,z1,Marcador_TCP\WObj:=Caja_2;
        MoveL Target_160_2,v1000,z1,Marcador_TCP\WObj:=Caja_2;
        MoveL Target_170_2,v1000,z1,Marcador_TCP\WObj:=Caja_2;
        MoveL Target_180_2,v1000,z1,Marcador_TCP\WObj:=Caja_2;
        MoveL Target_190_2,v1000,z1,Marcador_TCP\WObj:=Caja_2;
        MoveL Target_200_2,v1000,z1,Marcador_TCP\WObj:=Caja_2;
        MoveL Target_210_2,v1000,z1,Marcador_TCP\WObj:=Caja_2;
        MoveL Target_220_2,v1000,z1,Marcador_TCP\WObj:=Caja_2;
        MoveL Target_230_2,v1000,z1,Marcador_TCP\WObj:=Caja_2;
        MoveL Target_240_2,v1000,z1,Marcador_TCP\WObj:=Caja_2;
        MoveL Target_250_2,v1000,z1,Marcador_TCP\WObj:=Caja_2;
        MoveL Target_260_2,v1000,z1,Marcador_TCP\WObj:=Caja_2;
        MoveL Target_270_2,v1000,z1,Marcador_TCP\WObj:=Caja_2;
        MoveL Target_280_2,v1000,z1,Marcador_TCP\WObj:=Caja_2;
        MoveL Target_290_2,v1000,z1,Marcador_TCP\WObj:=Caja_2;
        MoveL Target_300_2,v1000,z1,Marcador_TCP\WObj:=Caja_2;
        MoveL Target_310_2,v1000,z1,Marcador_TCP\WObj:=Caja_2;
        MoveL Target_320_2,v1000,z1,Marcador_TCP\WObj:=Caja_2;
        MoveL Target_330_2,v1000,z1,Marcador_TCP\WObj:=Caja_2;
        MoveL Target_340_2,v1000,z1,Marcador_TCP\WObj:=Caja_2;
        MoveL Target_350_2,v1000,z1,Marcador_TCP\WObj:=Caja_2;
        MoveL Target_360_2,v1000,z1,Marcador_TCP\WObj:=Caja_2;
        MoveL Target_370_2,v1000,z1,Marcador_TCP\WObj:=Caja_2;
        MoveL Target_380_2,v1000,z1,Marcador_TCP\WObj:=Caja_2;
        MoveL Target_390_2,v1000,z1,Marcador_TCP\WObj:=Caja_2;
        MoveL Target_400_2,v1000,z1,Marcador_TCP\WObj:=Caja_2;
        MoveL Target_410_2,v1000,z1,Marcador_TCP\WObj:=Caja_2;
        MoveL Target_420_2,v1000,z1,Marcador_TCP\WObj:=Caja_2;
        MoveL Target_430_2,v1000,z1,Marcador_TCP\WObj:=Caja_2;
        MoveL Target_440_2,v1000,z1,Marcador_TCP\WObj:=Caja_2;
        MoveL Target_450_2,v1000,z1,Marcador_TCP\WObj:=Caja_2;
        MoveL Target_460_2,v1000,z1,Marcador_TCP\WObj:=Caja_2;
        MoveL Target_470_2,v1000,z1,Marcador_TCP\WObj:=Caja_2;
        MoveL Target_480_2,v1000,z1,Marcador_TCP\WObj:=Caja_2;
        MoveL Target_490_2,v1000,z1,Marcador_TCP\WObj:=Caja_2;
        MoveL Target_500_2,v1000,z1,Marcador_TCP\WObj:=Caja_2;
        MoveL Target_510_2,v1000,z1,Marcador_TCP\WObj:=Caja_2;
        MoveL Target_520_2,v1000,z1,Marcador_TCP\WObj:=Caja_2;
        MoveL Target_530_2,v1000,z1,Marcador_TCP\WObj:=Caja_2;
        MoveL Target_540_2,v1000,z1,Marcador_TCP\WObj:=Caja_2;
        MoveL Target_550_2,v1000,z1,Marcador_TCP\WObj:=Caja_2;
        MoveL Target_560_2,v1000,z1,Marcador_TCP\WObj:=Caja_2;
        MoveL Target_570_2,v1000,z1,Marcador_TCP\WObj:=Caja_2;
        MoveL Target_580_2,v1000,z1,Marcador_TCP\WObj:=Caja_2;
        MoveL Target_590_2,v1000,z1,Marcador_TCP\WObj:=Caja_2;
        MoveL Target_600_2,v1000,z1,Marcador_TCP\WObj:=Caja_2;
        MoveL Target_610_2,v1000,z1,Marcador_TCP\WObj:=Caja_2;
        MoveL Target_620_2,v1000,z1,Marcador_TCP\WObj:=Caja_2;
        MoveL Target_630_2,v1000,z1,Marcador_TCP\WObj:=Caja_2;
        MoveL Target_640_2,v1000,z1,Marcador_TCP\WObj:=Caja_2;
        MoveL Target_650_2,v1000,z1,Marcador_TCP\WObj:=Caja_2;
        MoveL Target_660_2,v1000,z1,Marcador_TCP\WObj:=Caja_2;
        MoveL Target_670_2,v1000,z1,Marcador_TCP\WObj:=Caja_2;
        MoveL Target_680_2,v1000,z1,Marcador_TCP\WObj:=Caja_2;
        MoveL Target_690_2,v1000,z1,Marcador_TCP\WObj:=Caja_2;
        MoveL Target_700_2,v1000,z1,Marcador_TCP\WObj:=Caja_2;
        MoveL Target_710_2,v1000,z1,Marcador_TCP\WObj:=Caja_2;
        MoveL Target_720_2,v1000,z1,Marcador_TCP\WObj:=Caja_2;
        MoveL Target_730_2,v1000,z1,Marcador_TCP\WObj:=Caja_2;
        MoveL Target_740_2,v1000,z1,Marcador_TCP\WObj:=Caja_2;
        MoveL Target_750_2,v1000,z1,Marcador_TCP\WObj:=Caja_2;
        MoveL Target_760_2,v1000,z1,Marcador_TCP\WObj:=Caja_2;
        MoveL Target_770_2,v1000,z1,Marcador_TCP\WObj:=Caja_2;
        MoveL Target_780_2,v1000,z1,Marcador_TCP\WObj:=Caja_2;
        MoveL Target_790_2,v1000,z1,Marcador_TCP\WObj:=Caja_2;
        MoveL Target_800_2,v1000,z1,Marcador_TCP\WObj:=Caja_2;
        MoveL Target_810_2,v1000,z1,Marcador_TCP\WObj:=Caja_2;
        MoveL Target_820_2,v1000,z1,Marcador_TCP\WObj:=Caja_2;
        MoveL Target_830_2,v1000,z1,Marcador_TCP\WObj:=Caja_2;
        MoveL Target_840_2,v1000,z1,Marcador_TCP\WObj:=Caja_2;
        MoveL Target_850_2,v1000,z1,Marcador_TCP\WObj:=Caja_2;
        MoveL Target_860_2,v1000,z1,Marcador_TCP\WObj:=Caja_2;
        MoveL Target_870_2,v1000,z1,Marcador_TCP\WObj:=Caja_2;
        MoveL Target_880_2,v1000,z1,Marcador_TCP\WObj:=Caja_2;
        MoveL Target_890_2,v1000,z1,Marcador_TCP\WObj:=Caja_2;
        MoveL Target_900_2,v1000,z1,Marcador_TCP\WObj:=Caja_2;
        MoveL Target_910_2,v1000,z1,Marcador_TCP\WObj:=Caja_2;
        MoveL Target_920_2,v1000,z1,Marcador_TCP\WObj:=Caja_2;
        MoveL Target_930_2,v1000,z1,Marcador_TCP\WObj:=Caja_2;
        MoveL Target_940_2,v1000,z1,Marcador_TCP\WObj:=Caja_2;
        MoveL Target_950_2,v1000,z1,Marcador_TCP\WObj:=Caja_2;
        MoveL Target_960_2,v1000,z1,Marcador_TCP\WObj:=Caja_2;
        MoveL Target_970_2,v1000,z1,Marcador_TCP\WObj:=Caja_2;
        MoveL Target_980_2,v1000,z1,Marcador_TCP\WObj:=Caja_2;
        MoveL Target_990_2,v1000,z1,Marcador_TCP\WObj:=Caja_2;
        MoveL Target_1000_2,v1000,z1,Marcador_TCP\WObj:=Caja_2;
        MoveL Target_1010_2,v1000,z1,Marcador_TCP\WObj:=Caja_2;
        MoveL Target_1020_2,v1000,z1,Marcador_TCP\WObj:=Caja_2;
        MoveL Target_1030_2,v1000,z1,Marcador_TCP\WObj:=Caja_2;
        MoveL Target_1040_2,v1000,z1,Marcador_TCP\WObj:=Caja_2;
        MoveL Target_1050_2,v1000,z1,Marcador_TCP\WObj:=Caja_2;
        MoveL Target_1060_2,v1000,z1,Marcador_TCP\WObj:=Caja_2;
        MoveL Target_1070_2,v1000,z1,Marcador_TCP\WObj:=Caja_2;
        MoveL Target_1080_2,v1000,z1,Marcador_TCP\WObj:=Caja_2;
        MoveL Target_1090_2,v1000,z1,Marcador_TCP\WObj:=Caja_2;
        MoveL Target_1100_2,v1000,z1,Marcador_TCP\WObj:=Caja_2;
        MoveL Target_1110_2,v1000,z1,Marcador_TCP\WObj:=Caja_2;
        MoveL Target_1120_2,v1000,z1,Marcador_TCP\WObj:=Caja_2;
        MoveL Target_1130_2,v1000,z1,Marcador_TCP\WObj:=Caja_2;
        MoveL Target_1140_2,v1000,z1,Marcador_TCP\WObj:=Caja_2;
        MoveL Target_1150_2,v1000,z1,Marcador_TCP\WObj:=Caja_2;
        MoveL Target_1160_2,v1000,z1,Marcador_TCP\WObj:=Caja_2;
        MoveL Target_1170_2,v1000,z1,Marcador_TCP\WObj:=Caja_2;
        MoveL Target_1180_2,v1000,z1,Marcador_TCP\WObj:=Caja_2;
        MoveL Target_1190_2,v1000,z1,Marcador_TCP\WObj:=Caja_2;
        MoveL Target_1200_2,v1000,z1,Marcador_TCP\WObj:=Caja_2;
        MoveL Target_1210_2,v1000,z1,Marcador_TCP\WObj:=Caja_2;
        MoveL Target_1220_2,v1000,z1,Marcador_TCP\WObj:=Caja_2;
        MoveL Target_1230_2,v1000,z1,Marcador_TCP\WObj:=Caja_2;
        MoveL Target_1240_2,v1000,z1,Marcador_TCP\WObj:=Caja_2;
        MoveL Target_1250_2,v1000,z1,Marcador_TCP\WObj:=Caja_2;
        MoveL Target_1260_2,v1000,z1,Marcador_TCP\WObj:=Caja_2;
        MoveL Target_1270_2,v1000,z1,Marcador_TCP\WObj:=Caja_2;
        MoveL Target_1280_2,v1000,z1,Marcador_TCP\WObj:=Caja_2;
        MoveL Target_1290_2,v1000,z1,Marcador_TCP\WObj:=Caja_2;
        MoveL Target_1300_2,v1000,z1,Marcador_TCP\WObj:=Caja_2;
        MoveL Target_1310_2,v1000,z1,Marcador_TCP\WObj:=Caja_2;
        MoveL Target_1320_2,v1000,z1,Marcador_TCP\WObj:=Caja_2;
        MoveL Target_1330_2,v1000,z1,Marcador_TCP\WObj:=Caja_2;
        MoveL Target_1340_2,v1000,z1,Marcador_TCP\WObj:=Caja_2;
        MoveL Target_1350_2,v1000,z1,Marcador_TCP\WObj:=Caja_2;
        MoveL Target_1360_2,v1000,z1,Marcador_TCP\WObj:=Caja_2;
        MoveL Target_1370_2,v1000,z1,Marcador_TCP\WObj:=Caja_2;
        MoveL Target_1380_2,v1000,z1,Marcador_TCP\WObj:=Caja_2;
        MoveL Target_1390_2,v1000,z1,Marcador_TCP\WObj:=Caja_2;
        MoveL Target_1400_2,v1000,z1,Marcador_TCP\WObj:=Caja_2;
        MoveL Target_1410_2,v1000,z1,Marcador_TCP\WObj:=Caja_2;
        MoveL Target_1420_2,v1000,z1,Marcador_TCP\WObj:=Caja_2;
        MoveL Target_1430_2,v1000,z1,Marcador_TCP\WObj:=Caja_2;
        MoveL Target_1440_2,v1000,z1,Marcador_TCP\WObj:=Caja_2;
        MoveL Target_1450_2,v1000,z1,Marcador_TCP\WObj:=Caja_2;
        MoveL Target_1460_2,v1000,z1,Marcador_TCP\WObj:=Caja_2;
        MoveL Target_1470_2,v1000,z1,Marcador_TCP\WObj:=Caja_2;
        MoveL Target_1480_2,v1000,z1,Marcador_TCP\WObj:=Caja_2;
        MoveL Target_1490_2,v1000,z1,Marcador_TCP\WObj:=Caja_2;
        MoveL Target_1500_2,v1000,z1,Marcador_TCP\WObj:=Caja_2;
        MoveL Target_1510_2,v1000,z1,Marcador_TCP\WObj:=Caja_2;
        MoveL Target_1520_2,v1000,z1,Marcador_TCP\WObj:=Caja_2;
        MoveL Target_1530_2,v1000,z1,Marcador_TCP\WObj:=Caja_2;
        MoveL Target_1540_2,v1000,z1,Marcador_TCP\WObj:=Caja_2;
        MoveL Target_1550_2,v1000,z1,Marcador_TCP\WObj:=Caja_2;
        MoveL Target_1560_2,v1000,z1,Marcador_TCP\WObj:=Caja_2;
        MoveL Target_1570_2,v1000,z1,Marcador_TCP\WObj:=Caja_2;
        MoveL Target_1580_2,v1000,z1,Marcador_TCP\WObj:=Caja_2;
        MoveL Target_1590_2,v1000,z1,Marcador_TCP\WObj:=Caja_2;
        MoveL Target_1600_2,v1000,z1,Marcador_TCP\WObj:=Caja_2;
        MoveL Target_1610_2,v1000,z1,Marcador_TCP\WObj:=Caja_2;
        MoveL Target_1620_2,v1000,z1,Marcador_TCP\WObj:=Caja_2;
        MoveL Target_1630_2,v1000,z1,Marcador_TCP\WObj:=Caja_2;
        MoveL Target_1640_2,v1000,z1,Marcador_TCP\WObj:=Caja_2;
        MoveL Target_1650_2,v1000,z1,Marcador_TCP\WObj:=Caja_2;
        MoveL Target_1660_2,v1000,z1,Marcador_TCP\WObj:=Caja_2;
        MoveL Target_1670_2,v1000,z1,Marcador_TCP\WObj:=Caja_2;
        MoveL Target_1680_2,v1000,z1,Marcador_TCP\WObj:=Caja_2;
        MoveL Target_1690_2,v1000,z1,Marcador_TCP\WObj:=Caja_2;
        MoveL Target_1700_2,v1000,z1,Marcador_TCP\WObj:=Caja_2;
        MoveL Target_1710_2,v1000,z1,Marcador_TCP\WObj:=Caja_2;
        MoveL Target_1720_2,v1000,z1,Marcador_TCP\WObj:=Caja_2;
        MoveL Target_1730_2,v1000,z1,Marcador_TCP\WObj:=Caja_2;
        MoveL Target_1740_2,v1000,z1,Marcador_TCP\WObj:=Caja_2;
        MoveL Target_1750_2,v1000,z1,Marcador_TCP\WObj:=Caja_2;
        MoveL Target_1760_2,v1000,z1,Marcador_TCP\WObj:=Caja_2;
        MoveL Target_1770_2,v1000,z1,Marcador_TCP\WObj:=Caja_2;
        MoveL Target_1780_2,v1000,z1,Marcador_TCP\WObj:=Caja_2;
        MoveL Target_1790_2,v1000,z1,Marcador_TCP\WObj:=Caja_2;
        MoveL Target_1800_2,v1000,z1,Marcador_TCP\WObj:=Caja_2;
        MoveL Target_1810_2,v1000,z1,Marcador_TCP\WObj:=Caja_2;
        MoveL Target_1820_2,v1000,z1,Marcador_TCP\WObj:=Caja_2;
        MoveL Target_1830_2,v1000,z1,Marcador_TCP\WObj:=Caja_2;
        MoveL Target_1840_2,v1000,z1,Marcador_TCP\WObj:=Caja_2;
        MoveL Target_1850_2,v1000,z1,Marcador_TCP\WObj:=Caja_2;
        MoveL Target_1860_2,v1000,z1,Marcador_TCP\WObj:=Caja_2;
        MoveL Target_1870_2,v1000,z1,Marcador_TCP\WObj:=Caja_2;
        MoveL Target_1880_2,v1000,z1,Marcador_TCP\WObj:=Caja_2;
        MoveL Target_1890_2,v1000,z1,Marcador_TCP\WObj:=Caja_2;
        MoveL Target_1900_2,v1000,z1,Marcador_TCP\WObj:=Caja_2;
        MoveL Target_1910_2,v1000,z1,Marcador_TCP\WObj:=Caja_2;
        MoveL Target_1920_2,v1000,z1,Marcador_TCP\WObj:=Caja_2;
        MoveL Target_1930_2,v1000,z1,Marcador_TCP\WObj:=Caja_2;
        MoveL Target_1940_2,v1000,z1,Marcador_TCP\WObj:=Caja_2;
        MoveL Target_1950_2,v1000,z1,Marcador_TCP\WObj:=Caja_2;
        MoveL Target_1960_2,v1000,z1,Marcador_TCP\WObj:=Caja_2;
        MoveL Target_1970_2,v1000,z1,Marcador_TCP\WObj:=Caja_2;
        MoveL Target_1980_2,v1000,z1,Marcador_TCP\WObj:=Caja_2;
        MoveL Target_1990_2,v1000,z1,Marcador_TCP\WObj:=Caja_2;
        MoveL Target_2000_2,v1000,z1,Marcador_TCP\WObj:=Caja_2;
        MoveL Target_2010_2,v1000,z1,Marcador_TCP\WObj:=Caja_2;
        MoveL Target_2020_2,v1000,z1,Marcador_TCP\WObj:=Caja_2;
        MoveL Target_2030_2,v1000,z1,Marcador_TCP\WObj:=Caja_2;
        MoveL Target_2040_2,v1000,z1,Marcador_TCP\WObj:=Caja_2;
        MoveL Target_2050_2,v1000,z1,Marcador_TCP\WObj:=Caja_2;
        MoveL Target_2060_2,v1000,z1,Marcador_TCP\WObj:=Caja_2;
        MoveL Target_2070_2,v1000,z1,Marcador_TCP\WObj:=Caja_2;
        MoveL Target_2080_2,v1000,z1,Marcador_TCP\WObj:=Caja_2;
        MoveL Target_2090_2,v1000,z1,Marcador_TCP\WObj:=Caja_2;
        MoveL Target_2100_2,v1000,z1,Marcador_TCP\WObj:=Caja_2;
        MoveL Target_2110_2,v1000,z1,Marcador_TCP\WObj:=Caja_2;
        MoveL Target_2120_2,v1000,z1,Marcador_TCP\WObj:=Caja_2;
        MoveL Target_2130_2,v1000,z1,Marcador_TCP\WObj:=Caja_2;
        MoveL Target_2140_2,v1000,z1,Marcador_TCP\WObj:=Caja_2;
        MoveL Target_2150_2,v1000,z1,Marcador_TCP\WObj:=Caja_2;
        MoveL Target_2160_2,v1000,z1,Marcador_TCP\WObj:=Caja_2;
        MoveL Target_2170_2,v1000,z1,Marcador_TCP\WObj:=Caja_2;
        MoveL Target_2180_2,v1000,z1,Marcador_TCP\WObj:=Caja_2;
        MoveL Target_2190_2,v1000,z1,Marcador_TCP\WObj:=Caja_2;
        MoveL Target_2200_2,v1000,z1,Marcador_TCP\WObj:=Caja_2;
        MoveL Target_2210_2,v1000,z1,Marcador_TCP\WObj:=Caja_2;
        MoveL Target_2220_2,v1000,z1,Marcador_TCP\WObj:=Caja_2;
        MoveL Target_2230_2,v1000,z1,Marcador_TCP\WObj:=Caja_2;
        MoveL Target_2240_2,v1000,z1,Marcador_TCP\WObj:=Caja_2;
        MoveL Target_2250_2,v1000,z1,Marcador_TCP\WObj:=Caja_2;
        MoveL Target_2260_2,v1000,z1,Marcador_TCP\WObj:=Caja_2;
        MoveL Target_2270_2,v1000,z1,Marcador_TCP\WObj:=Caja_2;
        MoveL Target_2280_2,v1000,z1,Marcador_TCP\WObj:=Caja_2;
        MoveL Target_2290_2,v1000,z1,Marcador_TCP\WObj:=Caja_2;
        MoveL Target_2300_2,v1000,z1,Marcador_TCP\WObj:=Caja_2;
        MoveL Target_2310_2,v1000,z1,Marcador_TCP\WObj:=Caja_2;
        MoveL Target_2320_2,v1000,z1,Marcador_TCP\WObj:=Caja_2;
        MoveL Target_2330_2,v1000,z1,Marcador_TCP\WObj:=Caja_2;
        MoveL Target_2340_2,v1000,z1,Marcador_TCP\WObj:=Caja_2;
        MoveL Target_2350_2,v1000,z1,Marcador_TCP\WObj:=Caja_2;
        MoveL Target_2360_2,v1000,z1,Marcador_TCP\WObj:=Caja_2;
        MoveL Target_2370_2,v1000,z1,Marcador_TCP\WObj:=Caja_2;
        MoveL Target_2380_2,v1000,z1,Marcador_TCP\WObj:=Caja_2;
        MoveL Target_2390_2,v1000,z1,Marcador_TCP\WObj:=Caja_2;
        MoveL Target_2400_2,v1000,z1,Marcador_TCP\WObj:=Caja_2;
        MoveL Target_2410_2,v1000,z1,Marcador_TCP\WObj:=Caja_2;
        MoveL Target_2420_2,v1000,z1,Marcador_TCP\WObj:=Caja_2;
        MoveL Target_2430_2,v1000,z1,Marcador_TCP\WObj:=Caja_2;
        MoveL Target_2440_2,v1000,z1,Marcador_TCP\WObj:=Caja_2;
        MoveL Target_2450_2,v1000,z1,Marcador_TCP\WObj:=Caja_2;
        MoveL Target_2460_2,v1000,z1,Marcador_TCP\WObj:=Caja_2;
        MoveL Target_2470_2,v1000,z1,Marcador_TCP\WObj:=Caja_2;
        MoveL Target_2480_2,v1000,z1,Marcador_TCP\WObj:=Caja_2;
        MoveL Target_2490_2,v1000,z1,Marcador_TCP\WObj:=Caja_2;
        MoveL Target_2500_2,v1000,z1,Marcador_TCP\WObj:=Caja_2;
        MoveL Target_2510_2,v1000,z1,Marcador_TCP\WObj:=Caja_2;
        MoveL Target_2520_2,v1000,z1,Marcador_TCP\WObj:=Caja_2;
        MoveL Target_2530_2,v1000,z1,Marcador_TCP\WObj:=Caja_2;
        MoveL Target_2540_2,v1000,z1,Marcador_TCP\WObj:=Caja_2;
        MoveL Target_2550_2,v1000,z1,Marcador_TCP\WObj:=Caja_2;
        MoveL Target_2560_2,v1000,z1,Marcador_TCP\WObj:=Caja_2;
        MoveL Target_2570_2,v1000,z1,Marcador_TCP\WObj:=Caja_2;
        MoveL Target_2580_2,v1000,z1,Marcador_TCP\WObj:=Caja_2;
        MoveL Target_2590_2,v1000,z1,Marcador_TCP\WObj:=Caja_2;
        MoveL Target_2600_2,v1000,z1,Marcador_TCP\WObj:=Caja_2;
        MoveL Target_2610_2,v1000,z1,Marcador_TCP\WObj:=Caja_2;
        MoveL Target_2620_2,v1000,z1,Marcador_TCP\WObj:=Caja_2;
        MoveL Target_2630_2,v1000,z1,Marcador_TCP\WObj:=Caja_2;
        MoveL Target_2640_2,v1000,z1,Marcador_TCP\WObj:=Caja_2;
        MoveL Target_2650_2,v1000,z1,Marcador_TCP\WObj:=Caja_2;
        MoveL Target_2660_2,v1000,z1,Marcador_TCP\WObj:=Caja_2;
        MoveL Target_2670_2,v1000,z1,Marcador_TCP\WObj:=Caja_2;
        MoveL Target_2680_2,v1000,z1,Marcador_TCP\WObj:=Caja_2;
        MoveL Target_2690_2,v1000,z1,Marcador_TCP\WObj:=Caja_2;
        MoveL Target_2700_2,v1000,z1,Marcador_TCP\WObj:=Caja_2;
        MoveL Target_2710_2,v1000,z1,Marcador_TCP\WObj:=Caja_2;
        MoveL Target_2720_2,v1000,z1,Marcador_TCP\WObj:=Caja_2;
        MoveL Target_2730_2,v1000,z1,Marcador_TCP\WObj:=Caja_2;
        MoveL Target_2740_2,v1000,z1,Marcador_TCP\WObj:=Caja_2;
        MoveL Target_2750_2,v1000,z1,Marcador_TCP\WObj:=Caja_2;
        MoveL Target_2760_2,v1000,z1,Marcador_TCP\WObj:=Caja_2;
        MoveL Target_2770_2,v1000,z1,Marcador_TCP\WObj:=Caja_2;
        MoveL Target_2780_2,v1000,z1,Marcador_TCP\WObj:=Caja_2;
        MoveL Target_2790_2,v1000,z1,Marcador_TCP\WObj:=Caja_2;
        MoveL Target_2800_2,v1000,z1,Marcador_TCP\WObj:=Caja_2;
        MoveL Target_2810_2,v1000,z1,Marcador_TCP\WObj:=Caja_2;
        MoveL Target_2820_2,v1000,z1,Marcador_TCP\WObj:=Caja_2;
        MoveL Target_2830_2,v1000,z1,Marcador_TCP\WObj:=Caja_2;
        MoveL Target_2840_2,v1000,z1,Marcador_TCP\WObj:=Caja_2;
        MoveL Target_2850_2,v1000,z1,Marcador_TCP\WObj:=Caja_2;
        MoveL Target_2860_2,v1000,z1,Marcador_TCP\WObj:=Caja_2;
        MoveL Target_2870_2,v1000,z1,Marcador_TCP\WObj:=Caja_2;
        MoveL Target_2880_2,v1000,z1,Marcador_TCP\WObj:=Caja_2;
        MoveL Target_2890_2,v1000,z1,Marcador_TCP\WObj:=Caja_2;
        MoveL Target_2900_2,v1000,z1,Marcador_TCP\WObj:=Caja_2;
        MoveL Target_2910_2,v1000,z1,Marcador_TCP\WObj:=Caja_2;
        MoveL Target_2920_2,v1000,z1,Marcador_TCP\WObj:=Caja_2;
        MoveL Target_2930_2,v1000,z1,Marcador_TCP\WObj:=Caja_2;
        MoveL Target_2940_2,v1000,z1,Marcador_TCP\WObj:=Caja_2;
        MoveL Target_2950_2,v1000,z1,Marcador_TCP\WObj:=Caja_2;
        MoveL Target_2960_2,v1000,z1,Marcador_TCP\WObj:=Caja_2;
        MoveL Target_2970_2,v1000,z1,Marcador_TCP\WObj:=Caja_2;
        MoveL Target_2980_2,v1000,z1,Marcador_TCP\WObj:=Caja_2;
        MoveL Target_2990_2,v1000,z1,Marcador_TCP\WObj:=Caja_2;
        MoveL Target_3000_2,v1000,z1,Marcador_TCP\WObj:=Caja_2;
        MoveL Target_3010_2,v1000,z1,Marcador_TCP\WObj:=Caja_2;
        MoveL Target_3020_2,v1000,z1,Marcador_TCP\WObj:=Caja_2;
        MoveL Target_3030_2,v1000,z1,Marcador_TCP\WObj:=Caja_2;
        MoveL Target_3040_2,v1000,z1,Marcador_TCP\WObj:=Caja_2;
        MoveL Target_3050_2,v1000,z1,Marcador_TCP\WObj:=Caja_2;
        MoveL Target_3060_2,v1000,z1,Marcador_TCP\WObj:=Caja_2;
        MoveL Target_3070_2,v1000,z1,Marcador_TCP\WObj:=Caja_2;
        MoveL Target_3080_2,v1000,z1,Marcador_TCP\WObj:=Caja_2;
        MoveL Target_3090_2,v1000,z1,Marcador_TCP\WObj:=Caja_2;
        MoveL Target_3100_2,v1000,z1,Marcador_TCP\WObj:=Caja_2;
        MoveL Target_3110_2,v1000,z1,Marcador_TCP\WObj:=Caja_2;
        MoveL Target_3120_2,v1000,z1,Marcador_TCP\WObj:=Caja_2;
        MoveL Target_3130_2,v1000,z1,Marcador_TCP\WObj:=Caja_2;
        MoveL Target_3140_2,v1000,z1,Marcador_TCP\WObj:=Caja_2;
        MoveL Target_3150_2,v1000,z1,Marcador_TCP\WObj:=Caja_2;
        MoveL Target_3160_2,v1000,z1,Marcador_TCP\WObj:=Caja_2;
        MoveL Target_3170_2,v1000,z1,Marcador_TCP\WObj:=Caja_2;
        MoveL Target_3180_2,v1000,z1,Marcador_TCP\WObj:=Caja_2;
        MoveL Target_3190_2,v1000,z1,Marcador_TCP\WObj:=Caja_2;
        MoveL Target_3200_2,v1000,z1,Marcador_TCP\WObj:=Caja_2;
        MoveL Target_3210_2,v1000,z1,Marcador_TCP\WObj:=Caja_2;
        MoveL Target_3220_2,v1000,z1,Marcador_TCP\WObj:=Caja_2;
        MoveL Target_3230_2,v1000,z1,Marcador_TCP\WObj:=Caja_2;
        MoveL Target_3240_2,v1000,z1,Marcador_TCP\WObj:=Caja_2;
        MoveL Target_3250_2,v1000,z1,Marcador_TCP\WObj:=Caja_2;
        MoveL Target_3260_2,v1000,z1,Marcador_TCP\WObj:=Caja_2;
        MoveL Target_3270_2,v1000,z1,Marcador_TCP\WObj:=Caja_2;
        MoveL Target_3280_2,v1000,z1,Marcador_TCP\WObj:=Caja_2;
        MoveL Target_3290_2,v1000,z1,Marcador_TCP\WObj:=Caja_2;
        MoveL Target_3300_2,v1000,z1,Marcador_TCP\WObj:=Caja_2;
        MoveL Target_3310_2,v1000,z1,Marcador_TCP\WObj:=Caja_2;
        MoveL Target_3320_2,v1000,z1,Marcador_TCP\WObj:=Caja_2;
        MoveL Target_3330_2,v1000,z1,Marcador_TCP\WObj:=Caja_2;
        MoveL Target_3340_2,v1000,z1,Marcador_TCP\WObj:=Caja_2;
        MoveL Target_3350_2,v1000,z1,Marcador_TCP\WObj:=Caja_2;
        MoveL Target_3360_2,v1000,z1,Marcador_TCP\WObj:=Caja_2;
        MoveL Target_3370_2,v1000,z1,Marcador_TCP\WObj:=Caja_2;
        MoveL Target_3380_2,v1000,z1,Marcador_TCP\WObj:=Caja_2;
        MoveL Target_3390_2,v1000,z1,Marcador_TCP\WObj:=Caja_2;
        MoveL Target_3400_2,v1000,z1,Marcador_TCP\WObj:=Caja_2;
        MoveL Target_3410_2,v1000,z1,Marcador_TCP\WObj:=Caja_2;
        MoveL Target_3420_2,v1000,z1,Marcador_TCP\WObj:=Caja_2;
        MoveL Target_3430_2,v1000,z1,Marcador_TCP\WObj:=Caja_2;
        MoveL Target_3440_2,v1000,z1,Marcador_TCP\WObj:=Caja_2;
        MoveL Target_3450_2,v1000,z1,Marcador_TCP\WObj:=Caja_2;
        MoveL Target_3460_2,v1000,z1,Marcador_TCP\WObj:=Caja_2;
        MoveL Target_3470_2,v1000,z1,Marcador_TCP\WObj:=Caja_2;
        MoveL Target_3480_2,v1000,z1,Marcador_TCP\WObj:=Caja_2;
        MoveL Target_3490_2,v1000,z1,Marcador_TCP\WObj:=Caja_2;
        MoveL Target_3500_2,v1000,z1,Marcador_TCP\WObj:=Caja_2;
        MoveL Target_3510_2,v1000,z1,Marcador_TCP\WObj:=Caja_2;
        MoveL Target_3520_2,v1000,z1,Marcador_TCP\WObj:=Caja_2;
        MoveL Target_3530_2,v1000,z1,Marcador_TCP\WObj:=Caja_2;
        MoveL Target_3540_2,v1000,z1,Marcador_TCP\WObj:=Caja_2;
        MoveL Target_3550_2,v1000,z1,Marcador_TCP\WObj:=Caja_2;
        MoveL Target_3560_2,v1000,z1,Marcador_TCP\WObj:=Caja_2;
        MoveL Target_3570_2,v1000,z1,Marcador_TCP\WObj:=Caja_2;
        MoveL Target_3580_2,v1000,z1,Marcador_TCP\WObj:=Caja_2;
        MoveL Target_3590_2,v1000,z1,Marcador_TCP\WObj:=Caja_2;
        MoveL Target_3600_2,v1000,z1,Marcador_TCP\WObj:=Caja_2;
        MoveL Target_3610_2,v1000,z1,Marcador_TCP\WObj:=Caja_2;
        MoveL Target_3620_2,v1000,z1,Marcador_TCP\WObj:=Caja_2;
        MoveL Target_3630_2,v1000,z1,Marcador_TCP\WObj:=Caja_2;
        MoveL Target_3640_2,v1000,z1,Marcador_TCP\WObj:=Caja_2;
        MoveL Target_3650_2,v1000,z1,Marcador_TCP\WObj:=Caja_2;
        MoveL Target_3660_2,v1000,z1,Marcador_TCP\WObj:=Caja_2;
        MoveL Target_3670_2,v1000,z1,Marcador_TCP\WObj:=Caja_2;
        MoveL Target_3680_2,v1000,z1,Marcador_TCP\WObj:=Caja_2;
        MoveL Target_3690_2,v1000,z1,Marcador_TCP\WObj:=Caja_2;
        MoveL Target_3700_2,v1000,z1,Marcador_TCP\WObj:=Caja_2;
        MoveL Target_3710_2,v1000,z1,Marcador_TCP\WObj:=Caja_2;
        MoveL Target_3720_2,v1000,z1,Marcador_TCP\WObj:=Caja_2;
        MoveL Target_3730_2,v1000,z1,Marcador_TCP\WObj:=Caja_2;
        MoveL Target_3740_2,v1000,z1,Marcador_TCP\WObj:=Caja_2;
        MoveL Target_3750_2,v1000,z1,Marcador_TCP\WObj:=Caja_2;
        MoveL Target_3760_2,v1000,z1,Marcador_TCP\WObj:=Caja_2;
        MoveL Target_3770_2,v1000,z1,Marcador_TCP\WObj:=Caja_2;
        MoveL Target_3780_2,v1000,z1,Marcador_TCP\WObj:=Caja_2;
        MoveL Target_3790_2,v1000,z1,Marcador_TCP\WObj:=Caja_2;
        MoveL Target_3800_2,v1000,z1,Marcador_TCP\WObj:=Caja_2;
        MoveL Target_3810_2,v1000,z1,Marcador_TCP\WObj:=Caja_2;
        MoveL Target_3820_2,v1000,z1,Marcador_TCP\WObj:=Caja_2;
        MoveL Target_3830_2,v1000,z1,Marcador_TCP\WObj:=Caja_2;
        MoveL Target_3840_2,v1000,z1,Marcador_TCP\WObj:=Caja_2;
        MoveL Target_3850_2,v1000,z1,Marcador_TCP\WObj:=Caja_2;
        MoveL Target_3860_2,v1000,z1,Marcador_TCP\WObj:=Caja_2;
        MoveL Target_3870_2,v1000,z1,Marcador_TCP\WObj:=Caja_2;
        MoveL Target_3880_2,v1000,z1,Marcador_TCP\WObj:=Caja_2;
        MoveL Target_3890_2,v1000,z1,Marcador_TCP\WObj:=Caja_2;
        MoveL Target_3900_2,v1000,z1,Marcador_TCP\WObj:=Caja_2;
        MoveL Target_3910_2,v1000,z1,Marcador_TCP\WObj:=Caja_2;
        MoveL Target_3920_2,v1000,z1,Marcador_TCP\WObj:=Caja_2;
        MoveL Target_3930_2,v1000,z1,Marcador_TCP\WObj:=Caja_2;
        MoveL Target_3940_2,v1000,z1,Marcador_TCP\WObj:=Caja_2;
        MoveL Target_3950_2,v1000,z1,Marcador_TCP\WObj:=Caja_2;
        MoveL Target_3960_2,v1000,z1,Marcador_TCP\WObj:=Caja_2;
        MoveL Target_3970_2,v1000,z1,Marcador_TCP\WObj:=Caja_2;
        MoveL Target_3980_2,v1000,z1,Marcador_TCP\WObj:=Caja_2;
        MoveL Target_3990_2,v1000,z1,Marcador_TCP\WObj:=Caja_2;
        MoveL Target_4000_2,v1000,z1,Marcador_TCP\WObj:=Caja_2;
        MoveL Target_4010_2,v1000,z1,Marcador_TCP\WObj:=Caja_2;
        MoveL Target_4020_2,v1000,z1,Marcador_TCP\WObj:=Caja_2;
        MoveL Target_4030_2,v1000,z1,Marcador_TCP\WObj:=Caja_2;
        MoveL Target_4040_2,v1000,z1,Marcador_TCP\WObj:=Caja_2;
        MoveL Target_4050_2,v1000,z1,Marcador_TCP\WObj:=Caja_2;
        MoveL Home_cafe_2,v60,z100,Marcador_TCP\WObj:=Caja_2;
        MoveL Target_Home_Espejo,v1000,z1,Marcador_TCP\WObj:=Caja_2;
    ENDPROC
ENDMODULE
